(* CODESYS project MC516.project
   CompiledLibraryCompatibilityVersion: LeadSysStudio V3.5 SP15 Patch 4
   Title: MC516

Project tree, tasks and I/O mapping:
  Device : MC516, Leadshine Technology Co., Ltd., order no. 516101, version 3.5.15.40
      settings: RetainMode = 0; RetainStartAddr = 20480; RetainEndAddr = 524288; RetainSize = 524288
    application Application
      libraries: Standard, * (System)
      task EtherCAT_Master_Leadshine_A (cyclic, interval 2000 µs, priority 0) calls EtherCAT_Master_Leadshine_A.EtherCAT_Task, MAIN
      program MAIN [ST]: io, motion, save_check, save_apply, work
      DataMain/
        data type HMIData
        data type SaveData
      function block AxisFB [ST]
      Enum/
        data type State
      Object/
        data type Button
        data type Cylinder
        data type AxisEC
      function StateNext [ST]
      DataWork/
        data type SupplyData
        data type WorkData
        data type CutData
      function block CutFB [ST]
      visualisation Visualization
      function block SupplyFB [ST]
      Symbols
      global variables PersistentVars
    Resource Usage
    Device Diagnose
    Network Configuration
      LocalBus Config
    SoftMotion General Axis Pool
      JogEncoder : SMC_FreeEncoder, 3S - Smart Software Solutions GmbH, order no. 1805, version 3.5.5.0
          settings: wDriveID = 3; dwRatioTechUnitsDenom = 400; ScalingIncs = 400
    High_Speed_IO_Module : High Speed IO, Leadshine Technology Co., Ltd., version 3.5.15.40
        settings: HS_IO_Mode_0.High In IO Mode 0 = 196611; HS_IO_Mode_0.High In IO Mode 2 = 196611; Counter_Mask = 5; Ioin_Mask = 19; HS counter 1.Counter_CountMode = 1; HS counter 2.Counter_CountMode = 1; HS counter 3.Counter_SetWorkMode = 2; HS counter 3.Counter_CountMode = 1; InputFilter Para.Time_In0 = 2; InputFilter Para.Time_In1 = 2; InputFilter Para.Time_In4 = 2
        unmapped channels: Genral_IO_IN, Genral_IO_Out
    LocalBus_Master_Module : LocalBus Master, Leadshine Technology Co., Ltd., version 3.5.15.40
    EtherCAT_Master_Leadshine_A : EtherCAT Master SoftMotion, 3S - Smart Software Solutions GmbH, version 3.5.15.30
        settings: MasterCycleTime = 2000; NetworkName = 'ecat'; SelectNetworkByName = TRUE; SrcAddress1 = 10; SrcAddress2 = 889192738
      XINJE_DS5C1_CoE_Drive_Rev4_0 : XINJE-DS5C1 EtherCAT(CoE) Drive Rev4.0 v3.7.70, Xinje Electronics, Inc., order no. XINJE-DS5C1 CoE Drive Rev4.0, version Revision=16#20201207
          settings: Number of Inputs = 6; Number of Infos about Inputs = 6; StationAlias = 1; Sync.Length = 17; FMMU.Length = 17; DC sync0 cycletime = 2000; DC sync1 cycletime = 2000; Number of SDO = 4; Interpolation time period.Value = 2; RxTxPdo.NumberofEntries = 6; RxTxPdo.Index = 16#1A00; RxTxPdo.DependOnSlot = False; RxTxPdo.DependOnSlotGroup = False; RxTxPdo.OverwrittenByModule = False; Status Word.Offset = 0; Status Word.DependOnSlot = False; Status Word.DependOnSlotGroup = False; ActualPosition.Offset = 0; ActualPosition.DependOnSlot = False; ActualPosition.DependOnSlotGroup = False; Velocity actual value.Offset = 0; Velocity actual value.DependOnSlot = False; Velocity actual value.DependOnSlotGroup = False; ActualTorque.Offset = 0; ActualTorque.DependOnSlot = False; ActualTorque.DependOnSlotGroup = False; ModeOfOperationDisplay.Offset = 0; ModeOfOperationDisplay.DependOnSlot = False; ModeOfOperationDisplay.DependOnSlotGroup = False; Index = 16#5000; SubIndex = 0; Size = 32; Offset = 0; DependOnSlot = False; DependOnSlotGroup = False; Status Word.Default = ''; Status Word.Comment = ''; ActualPosition.Default = ''; ActualPosition.Comment = ''; Velocity actual value.Default = '';
            Velocity actual value.Comment = ''; ActualTorque.Default = ''; ActualTorque.Comment = ''; ModeOfOperationDisplay.Default = ''; ModeOfOperationDisplay.Comment = ''; Name = 'Encode Single Position'; DataType = 'DINT'; Default = ''; Comment = ''
          unmapped channels: Control Word, TargetPosition, TargetVelocity, TargetTorque, ModeOfOperation, Status Word, ActualPosition, Velocity actual value, ActualTorque, ModeOfOperationDisplay, Encode Single Position
        Axis : Axis, 3S - Smart Software Solutions GmbH, order no. 0, version 4.6.1.0
            settings: wDriveID = 0; dwRatioTechUnitsDenom = 16384; iRatioTechUnitsNum = -625; eRampType = 3; Number of pulses for one revolution = 131072; The displacement for one revolution of the workbench = 5000; Gear ratio molecule = 1; Gear ratio denominator = 1; ScalingIncs = 131072; InvertDirection = True; AdrOffset_8010 = 4; BitOffset_8010 = 0; BitLength_8010 = 16; Address_8010 = '%QW2'; Type_8010 = 'UINT'; AddressPointer_8010 = ADR(%QW2); AdrOffset_8020 = 8; BitOffset_8020 = 0; BitLength_8020 = 32; Address_8020 = '%QD2'; Type_8020 = 'DINT'; AddressPointer_8020 = ADR(%QD2); AdrOffset_8030 = 12; BitOffset_8030 = 0; BitLength_8030 = 32; Address_8030 = '%QD3'; Type_8030 = 'DINT'; AddressPointer_8030 = ADR(%QD3); AdrOffset_8040 = 16; BitOffset_8040 = 0; BitLength_8040 = 16; Address_8040 = '%QW8'; Type_8040 = 'INT'; AddressPointer_8040 = ADR(%QW8); AdrOffset_8050 = 18; BitOffset_8050 = 0; BitLength_8050 = 8; Address_8050 = '%QB18'; Type_8050 = 'SINT'; AddressPointer_8050 = ADR(%QB18);
              AdrOffset_8060 = 4294967295; BitOffset_8060 = 0; BitLength_8060 = 0; Address_8060 = ''; Type_8060 = ''; AddressPointer_8060 = 0; AdrOffset_8070 = 4294967295; BitOffset_8070 = 0; BitLength_8070 = 0; Address_8070 = ''; Type_8070 = ''; AddressPointer_8070 = 0; AdrOffset_8080 = 4294967295; BitOffset_8080 = 0; BitLength_8080 = 0; Address_8080 = ''; Type_8080 = ''; AddressPointer_8080 = 0; AdrOffset_8090 = 4294967295; BitOffset_8090 = 0; BitLength_8090 = 0; Address_8090 = ''; Type_8090 = ''; AddressPointer_8090 = 0; AdrOffset_8510 = 4; BitOffset_8510 = 0; BitLength_8510 = 16; Address_8510 = '%IW2'; Type_8510 = 'UINT'; AddressPointer_8510 = ADR(%IW2); AdrOffset_8520 = 8; BitOffset_8520 = 0; BitLength_8520 = 32; Address_8520 = '%ID2'; Type_8520 = 'DINT'; AddressPointer_8520 = ADR(%ID2); AdrOffset_8530 = 12; BitOffset_8530 = 0; BitLength_8530 = 32; Address_8530 = '%ID3';
              Type_8530 = 'DINT'; AddressPointer_8530 = ADR(%ID3); AdrOffset_8540 = 16; BitOffset_8540 = 0; BitLength_8540 = 16; Address_8540 = '%IW8'; Type_8540 = 'INT'; AddressPointer_8540 = ADR(%IW8); AdrOffset_8550 = 18; BitOffset_8550 = 0; BitLength_8550 = 8; Address_8550 = '%IB18'; Type_8550 = 'SINT'; AddressPointer_8550 = ADR(%IB18); AdrOffset_8560 = 4294967295; BitOffset_8560 = 0; BitLength_8560 = 0; Address_8560 = ''; Type_8560 = ''; AddressPointer_8560 = 0; AdrOffset_8570 = 4294967295; BitOffset_8570 = 0; BitLength_8570 = 0; Address_8570 = ''; Type_8570 = ''; AddressPointer_8570 = 0; AdrOffset_8580 = 4294967295; BitOffset_8580 = 0; BitLength_8580 = 0; Address_8580 = ''; Type_8580 = ''; AddressPointer_8580 = 0; AdrOffset_8590 = 4294967295; BitOffset_8590 = 0; BitLength_8590 = 0; Address_8590 = ''; Type_8590 = ''; AddressPointer_8590 = 0; AdrOffset_8600 = 4294967295; BitOffset_8600 = 0;
              BitLength_8600 = 0; Address_8600 = ''; Type_8600 = ''; AddressPointer_8600 = 0; AdrOffset_8600 = 4294967295; BitOffset_8600 = 0; BitLength_8600 = 0; Address_8610 = ''; Type_8610 = ''; AddressPointer_8610 = 0; AdrOffset_8620 = 4294967295; BitOffset_8620 = 0; BitLength_8620 = 0; Address_8620 = ''; Type_8620 = ''; AddressPointer_8620 = 0
      XINJE_DS5C1_CoE_Drive_Rev4_0_1 : XINJE-DS5C1 EtherCAT(CoE) Drive Rev4.0 v3.7.70, Xinje Electronics, Inc., order no. XINJE-DS5C1 CoE Drive Rev4.0, version Revision=16#20201207
          settings: Number of Inputs = 6; Number of Infos about Inputs = 6; StationAlias = 1; Optional = False; DeviceIdenticationADO = 0; DeviceIdenticationMode = 0; Sync.Length = 17; FMMU.Length = 17; DC sync0 cycletime = 2000; DC sync1 cycletime = 2000; Number of SDO = 4; Interpolation time period.Value = 2; RxTxPdo.NumberofEntries = 6; RxTxPdo.Index = 16#1A00; RxTxPdo.DependOnSlot = False; RxTxPdo.DependOnSlotGroup = False; RxTxPdo.OverwrittenByModule = False; Status Word.Offset = 0; Status Word.DependOnSlot = False; Status Word.DependOnSlotGroup = False; ActualPosition.Offset = 0; ActualPosition.DependOnSlot = False; ActualPosition.DependOnSlotGroup = False; Velocity actual value.Offset = 0; Velocity actual value.DependOnSlot = False; Velocity actual value.DependOnSlotGroup = False; ActualTorque.Offset = 0; ActualTorque.DependOnSlot = False; ActualTorque.DependOnSlotGroup = False; ModeOfOperationDisplay.Offset = 0; ModeOfOperationDisplay.DependOnSlot = False; ModeOfOperationDisplay.DependOnSlotGroup = False; Index = 16#5000; SubIndex = 0; Size = 32; Offset = 0; DependOnSlot = False; DependOnSlotGroup = False; Status Word.Default = ''; Status Word.Comment = '';
            ActualPosition.Default = ''; ActualPosition.Comment = ''; Velocity actual value.Default = ''; Velocity actual value.Comment = ''; ActualTorque.Default = ''; ActualTorque.Comment = ''; ModeOfOperationDisplay.Default = ''; ModeOfOperationDisplay.Comment = ''; Name = 'Encode Single Position'; DataType = 'DINT'; Default = ''; Comment = ''
          unmapped channels: Control Word, TargetPosition, TargetVelocity, TargetTorque, ModeOfOperation, Status Word, ActualPosition, Velocity actual value, ActualTorque, ModeOfOperationDisplay, Encode Single Position
        Axis_1 : Axis, 3S - Smart Software Solutions GmbH, order no. 0, version 4.6.1.0
            settings: dwRatioTechUnitsDenom = 16384; iRatioTechUnitsNum = -625; eRampType = 3; Number of pulses for one revolution = 131072; The displacement for one revolution of the workbench = 5000; Gear ratio molecule = 1; Gear ratio denominator = 1; ScalingIncs = 131072; InvertDirection = True; AdrOffset_8010 = 20; BitOffset_8010 = 0; BitLength_8010 = 16; Address_8010 = '%QW10'; Type_8010 = 'UINT'; AddressPointer_8010 = ADR(%QW10); AdrOffset_8020 = 24; BitOffset_8020 = 0; BitLength_8020 = 32; Address_8020 = '%QD6'; Type_8020 = 'DINT'; AddressPointer_8020 = ADR(%QD6); AdrOffset_8030 = 28; BitOffset_8030 = 0; BitLength_8030 = 32; Address_8030 = '%QD7'; Type_8030 = 'DINT'; AddressPointer_8030 = ADR(%QD7); AdrOffset_8040 = 32; BitOffset_8040 = 0; BitLength_8040 = 16; Address_8040 = '%QW16'; Type_8040 = 'INT'; AddressPointer_8040 = ADR(%QW16); AdrOffset_8050 = 34; BitOffset_8050 = 0; BitLength_8050 = 8; Address_8050 = '%QB34'; Type_8050 = 'SINT'; AddressPointer_8050 = ADR(%QB34); AdrOffset_8060 = 4294967295;
              BitOffset_8060 = 0; BitLength_8060 = 0; Address_8060 = ''; Type_8060 = ''; AddressPointer_8060 = 0; AdrOffset_8070 = 4294967295; BitOffset_8070 = 0; BitLength_8070 = 0; Address_8070 = ''; Type_8070 = ''; AddressPointer_8070 = 0; AdrOffset_8080 = 4294967295; BitOffset_8080 = 0; BitLength_8080 = 0; Address_8080 = ''; Type_8080 = ''; AddressPointer_8080 = 0; AdrOffset_8090 = 4294967295; BitOffset_8090 = 0; BitLength_8090 = 0; Address_8090 = ''; Type_8090 = ''; AddressPointer_8090 = 0; AdrOffset_8510 = 24; BitOffset_8510 = 0; BitLength_8510 = 16; Address_8510 = '%IW12'; Type_8510 = 'UINT'; AddressPointer_8510 = ADR(%IW12); AdrOffset_8520 = 28; BitOffset_8520 = 0; BitLength_8520 = 32; Address_8520 = '%ID7'; Type_8520 = 'DINT'; AddressPointer_8520 = ADR(%ID7); AdrOffset_8530 = 32; BitOffset_8530 = 0; BitLength_8530 = 32; Address_8530 = '%ID8'; Type_8530 = 'DINT';
              AddressPointer_8530 = ADR(%ID8); AdrOffset_8540 = 36; BitOffset_8540 = 0; BitLength_8540 = 16; Address_8540 = '%IW18'; Type_8540 = 'INT'; AddressPointer_8540 = ADR(%IW18); AdrOffset_8550 = 38; BitOffset_8550 = 0; BitLength_8550 = 8; Address_8550 = '%IB38'; Type_8550 = 'SINT'; AddressPointer_8550 = ADR(%IB38); AdrOffset_8560 = 4294967295; BitOffset_8560 = 0; BitLength_8560 = 0; Address_8560 = ''; Type_8560 = ''; AddressPointer_8560 = 0; AdrOffset_8570 = 4294967295; BitOffset_8570 = 0; BitLength_8570 = 0; Address_8570 = ''; Type_8570 = ''; AddressPointer_8570 = 0; AdrOffset_8580 = 4294967295; BitOffset_8580 = 0; BitLength_8580 = 0; Address_8580 = ''; Type_8580 = ''; AddressPointer_8580 = 0; AdrOffset_8590 = 4294967295; BitOffset_8590 = 0; BitLength_8590 = 0; Address_8590 = ''; Type_8590 = ''; AddressPointer_8590 = 0; AdrOffset_8600 = 4294967295; BitOffset_8600 = 0; BitLength_8600 = 0;
              Address_8600 = ''; Type_8600 = ''; AddressPointer_8600 = 0; AdrOffset_8600 = 4294967295; BitOffset_8600 = 0; BitLength_8600 = 0; Address_8610 = ''; Type_8610 = ''; AddressPointer_8610 = 0; AdrOffset_8620 = 4294967295; BitOffset_8620 = 0; BitLength_8620 = 0; Address_8620 = ''; Type_8620 = ''; AddressPointer_8620 = 0
      XINJE_DS5C1_CoE_Drive_Rev4_0_2 : XINJE-DS5C1 EtherCAT(CoE) Drive Rev4.0 v3.7.70, Xinje Electronics, Inc., order no. XINJE-DS5C1 CoE Drive Rev4.0, version Revision=16#20201207
          settings: Number of Inputs = 6; Number of Infos about Inputs = 6; StationAlias = 1; Optional = False; DeviceIdenticationADO = 0; DeviceIdenticationMode = 0; Sync.Length = 17; FMMU.Length = 17; DC sync0 cycletime = 2000; DC sync1 cycletime = 2000; Number of SDO = 7; Interpolation time period.Value = 2; RxTxPdo.NumberofEntries = 6; RxTxPdo.Index = 16#1A00; RxTxPdo.DependOnSlot = False; RxTxPdo.DependOnSlotGroup = False; RxTxPdo.OverwrittenByModule = False; Status Word.Offset = 0; Status Word.DependOnSlot = False; Status Word.DependOnSlotGroup = False; ActualPosition.Offset = 0; ActualPosition.DependOnSlot = False; ActualPosition.DependOnSlotGroup = False; Velocity actual value.Offset = 0; Velocity actual value.DependOnSlot = False; Velocity actual value.DependOnSlotGroup = False; ActualTorque.Offset = 0; ActualTorque.DependOnSlot = False; ActualTorque.DependOnSlotGroup = False; ModeOfOperationDisplay.Offset = 0; ModeOfOperationDisplay.DependOnSlot = False; ModeOfOperationDisplay.DependOnSlotGroup = False; Index = 16#5000; SubIndex = 0; Size = 32; Offset = 0; DependOnSlot = False; DependOnSlotGroup = False; Status Word.Default = ''; Status Word.Comment = '';
            ActualPosition.Default = ''; ActualPosition.Comment = ''; Velocity actual value.Default = ''; Velocity actual value.Comment = ''; ActualTorque.Default = ''; ActualTorque.Comment = ''; ModeOfOperationDisplay.Default = ''; ModeOfOperationDisplay.Comment = ''; Name = 'Encode Single Position'; DataType = 'DINT'; Default = ''; Comment = ''
          unmapped channels: Control Word, TargetPosition, TargetVelocity, TargetTorque, ModeOfOperation, Status Word, ActualPosition, Velocity actual value, ActualTorque, ModeOfOperationDisplay, Encode Single Position
        Axis_2 : Axis, 3S - Smart Software Solutions GmbH, order no. 0, version 4.6.1.0
            settings: wDriveID = 2; dwRatioTechUnitsDenom = 90112; iRatioTechUnitsNum = -5625; iMovementType = 0; fPositionPeriod = 360000; eRampType = 3; Number of pulses for one revolution = 131072; The displacement for one revolution of the workbench = 360000; Gear ratio molecule = 44; Gear ratio denominator = 1; ScalingIncs = 131072; ScalingMotorTurns2 = 44; InvertDirection = True; AdrOffset_8010 = 36; BitOffset_8010 = 0; BitLength_8010 = 16; Address_8010 = '%QW18'; Type_8010 = 'UINT'; AddressPointer_8010 = ADR(%QW18); AdrOffset_8020 = 40; BitOffset_8020 = 0; BitLength_8020 = 32; Address_8020 = '%QD10'; Type_8020 = 'DINT'; AddressPointer_8020 = ADR(%QD10); AdrOffset_8030 = 44; BitOffset_8030 = 0; BitLength_8030 = 32; Address_8030 = '%QD11'; Type_8030 = 'DINT'; AddressPointer_8030 = ADR(%QD11); AdrOffset_8040 = 48; BitOffset_8040 = 0; BitLength_8040 = 16; Address_8040 = '%QW24'; Type_8040 = 'INT'; AddressPointer_8040 = ADR(%QW24); AdrOffset_8050 = 50; BitOffset_8050 = 0; BitLength_8050 = 8;
              Address_8050 = '%QB50'; Type_8050 = 'SINT'; AddressPointer_8050 = ADR(%QB50); AdrOffset_8060 = 4294967295; BitOffset_8060 = 0; BitLength_8060 = 0; Address_8060 = ''; Type_8060 = ''; AddressPointer_8060 = 0; AdrOffset_8070 = 4294967295; BitOffset_8070 = 0; BitLength_8070 = 0; Address_8070 = ''; Type_8070 = ''; AddressPointer_8070 = 0; AdrOffset_8080 = 4294967295; BitOffset_8080 = 0; BitLength_8080 = 0; Address_8080 = ''; Type_8080 = ''; AddressPointer_8080 = 0; AdrOffset_8090 = 4294967295; BitOffset_8090 = 0; BitLength_8090 = 0; Address_8090 = ''; Type_8090 = ''; AddressPointer_8090 = 0; AdrOffset_8510 = 44; BitOffset_8510 = 0; BitLength_8510 = 16; Address_8510 = '%IW22'; Type_8510 = 'UINT'; AddressPointer_8510 = ADR(%IW22); AdrOffset_8520 = 48; BitOffset_8520 = 0; BitLength_8520 = 32; Address_8520 = '%ID12'; Type_8520 = 'DINT'; AddressPointer_8520 = ADR(%ID12); AdrOffset_8530 = 52;
              BitOffset_8530 = 0; BitLength_8530 = 32; Address_8530 = '%ID13'; Type_8530 = 'DINT'; AddressPointer_8530 = ADR(%ID13); AdrOffset_8540 = 56; BitOffset_8540 = 0; BitLength_8540 = 16; Address_8540 = '%IW28'; Type_8540 = 'INT'; AddressPointer_8540 = ADR(%IW28); AdrOffset_8550 = 58; BitOffset_8550 = 0; BitLength_8550 = 8; Address_8550 = '%IB58'; Type_8550 = 'SINT'; AddressPointer_8550 = ADR(%IB58); AdrOffset_8560 = 4294967295; BitOffset_8560 = 0; BitLength_8560 = 0; Address_8560 = ''; Type_8560 = ''; AddressPointer_8560 = 0; AdrOffset_8570 = 4294967295; BitOffset_8570 = 0; BitLength_8570 = 0; Address_8570 = ''; Type_8570 = ''; AddressPointer_8570 = 0; AdrOffset_8580 = 4294967295; BitOffset_8580 = 0; BitLength_8580 = 0; Address_8580 = ''; Type_8580 = ''; AddressPointer_8580 = 0; AdrOffset_8590 = 4294967295; BitOffset_8590 = 0; BitLength_8590 = 0; Address_8590 = ''; Type_8590 = '';
              AddressPointer_8590 = 0; AdrOffset_8600 = 4294967295; BitOffset_8600 = 0; BitLength_8600 = 0; Address_8600 = ''; Type_8600 = ''; AddressPointer_8600 = 0; AdrOffset_8600 = 4294967295; BitOffset_8600 = 0; BitLength_8600 = 0; Address_8610 = ''; Type_8610 = ''; AddressPointer_8610 = 0; AdrOffset_8620 = 4294967295; BitOffset_8620 = 0; BitLength_8620 = 0; Address_8620 = ''; Type_8620 = ''; AddressPointer_8620 = 0
  text list GlobalTextList
*)

// Device/Application/DataMain/HMIData
{ attribute 'pack_mode' := ''}
TYPE HMIData :
STRUCT
	//
	save_data: SaveData;
	save: BOOL;
	save_need_check: BOOL;
	save_need: BOOL;
	//
	plc_ready: BOOL;
	hmi_ready: BOOL;
	run: BOOL;
	stop: BOOL;
	home: BOOL;
	overload_fixed: BOOL;
	foil_stuck_fix: BOOL;
	//
	supply_test: BOOL;
	supply_arm_clamp_holder: BOOL;
	supply_arm_clamp: BOOL;
	supply_spindle_clamp: BOOL;
	supply_spindle_extract: BOOL;
	supply_feeder_small: BOOL;
	supply_feeder_linear: BOOL;
	supply_feeder_big: BOOL;
	supply_feeder_test: BOOL;
	cut_spindle_run: BOOL;
	hydraulic_run: BOOL;
	jog_micro_per_rev: UINT;
	//
	view_input_run: BOOL;
	view_input_stop: BOOL;
	view_input_air: BOOL;
	view_input_hydraulic: BOOL;
	view_input_arm_clamp_holder_p: BOOL;
	view_input_feeder_small: BOOL;
	view_input_feeder_big: BOOL;
	view_input_jog_counter_a: BOOL;
	view_input_jog_counter_b: BOOL;
	view_input_jog_index_a: BOOL;
	view_input_jog_index_b: BOOL;
	view_input_spindle_encoder: BOOL;
	view_input_jog_index: UINT;
	view_input_jog_micro: DINT;
	//
	view_output_arm_clamp_holder: BOOL;
	view_output_arm_clamp: BOOL;
	view_output_spindle: BOOL;
	view_output_spindle_clamp_n: BOOL;
	view_output_spindle_clamp_p: BOOL;
	view_output_spindle_extract: BOOL;
	view_output_hydraulic: BOOL;
	view_output_alarm: BOOL;
	view_output_feeder_small: BOOL;
	view_output_feeder_linear: BOOL;
	view_output_feeder_big: BOOL;
	//
	view_can_run: BOOL;
	view_can_stop: BOOL;
	view_can_home: BOOL;
	view_run_auto: BOOL;
	view_manual_active: BOOL;
	//
	view_axiss_position_micron: ARRAY[0..2] OF UDINT;
	view_axiss_torque_mNm: ARRAY[0..2] OF UDINT;
	view_cut_spindle_run_ing: BOOL;
	view_cut_spindle_rpm: UDINT;
	//
	view_supply_test: ARRAY[0..4] OF BOOL;
	//
	view_overload: BOOL;
	view_supply_foil_short: BOOL;
	view_supply_foil_stuck: BOOL;
	view_cycle_count: UDINT;
	view_cycle_time_msec: UDINT;
	//
	view_state_work: INT;
	view_state_supply: INT;
	view_state_cut: INT;
	view_state_cut_spindle: INT;
END_STRUCT
END_TYPE

// Device/Application/DataMain/SaveData
{ attribute 'pack_mode' := ''}
TYPE SaveData :
STRUCT
	set_done: BOOL;
	//
	supply_begin_micro_deg: UDINT;
	supply_mid_micro_deg: UDINT;
	supply_end_micro_deg: UDINT;
	supply_micro_deg_per_sec: UDINT;
	//
	supply_arm_clamp_holder_n_delay_msec: UINT;
	supply_arm_clamp_holder_p_delay_msec: UINT;
	supply_arm_clamp_n_delay_msec: UINT;
	supply_arm_clamp_p_delay_msec: UINT;
	supply_spindle_clamp_n_delay_msec: UINT;
	supply_spindle_clamp_p_delay_msec: UINT;
	supply_spindle_extract_n_delay_msec: UINT;
	supply_spindle_extract_p_delay_msec: UINT;
	//
	cut_begin_micron: ARRAY[0..1] OF UDINT;
	cut_rapid_micron: ARRAY[0..1] OF UDINT;
	cut_end_micron: ARRAY[0..1] OF UDINT;
	cut_offset_micron: ARRAY[0..1] OF DINT;
	cut_lag_micron: UDINT;
	cut_rapid_micron_per_rev: UDINT;
	cut_micron_per_rev: UDINT;
	cut_dwell_msec: UINT;
	cut_retract_micron: UDINT; // vị trí lùi về
	cut_retract_micron_per_sec: UDINT; // tốc độ lùi sau khi cắt
	cut_spindle_encoder_resolution: UINT;
	//
	home_encoder_value_recorded: BOOL;
	home_encoder_value: ARRAY[0..2] OF DINT;
END_STRUCT
END_TYPE

// Device/Application/Enum/State
{attribute 'qualified_only'}
{attribute 'strict'}
TYPE State :
(
	NONE := 0,
	RST := 1,
	RST_DONE := 50,
	HOME := 51,
	HOME_FORWARD := 71,
	HOME_DONE := 90,
	HOME_OFFSET := 91,
	HOME_OFFSET_DONE := 99,
	READY := 100,
	RUN := 101,
	RUN_ING := 200
);
END_TYPE

// Device/Application/Object/Button
{ attribute 'pack_mode' := ''}
TYPE Button :
STRUCT
	on: BOOL;
	rise: R_TRIG;
	rise_physical: R_TRIG;
	fall: F_TRIG;
	fall_physical: F_TRIG;
	timer: TON;
END_STRUCT
END_TYPE

// Device/Application/Object/Cylinder
{ attribute 'pack_mode' := ''}
TYPE Cylinder :
STRUCT
	on: BOOL;
	n_timer: TON;
	p_timer: TON;
END_STRUCT
END_TYPE

// Device/Application/Object/AxisEC
{ attribute 'pack_mode' := ''}
TYPE AxisEC :
STRUCT
	///////
	//REF//
	///////
	ref: POINTER TO SM3_Drive_ETC_DS402_CyclicSync.AXIS_REF_ETC_DS402_CS;
	read: POINTER TO SMC3_ETC_ReadParameter_CoE;
	write: POINTER TO SMC3_ETC_WriteParameter_CoE;
	read_status: POINTER TO MC_ReadStatus;
	set_mode: POINTER TO SMC_SetControllerMode;
	power: POINTER TO MC_Power;
	reset: POINTER TO MC_Reset;
	stop: POINTER TO MC_Stop;
	inch: POINTER TO SMC_Inch;
	fsv: POINTER TO SMC_FollowSetValues;
	sp: POINTER TO MC_SetPosition;
	mabs: POINTER TO MC_MoveAbsolute;
	////////
	//DATA//
	////////
	encoder_resolution: DINT;
	torque_rated_Nm: LREAL;
	encoder_single_position: DINT;
	///////////
	//PROCESS//
	///////////
	state: INT;
	torque_Nm: LREAL;
	torque_Nm_abs: LREAL;
	overload: BOOL;
	overload_check: BOOL;
	overload_timer: TON;
	//home
	home_done: BOOL; // = TRUE khi về gốc thành công, chỉ về gốc khi bật máy
	home_torque_Nm: LREAL;
	home_hit_timer: TON;
	home_offset_absolute_μ: LREAL; // vị trí từ điểm va chạm đến gốc tuyệt đối, xem hàm save_apply()
	home_back_μ_per_sec: LREAL; // tốc độ lùi về lấy gốc
	home_forward_μ_per_sec: LREAL; // tốc độ tiến sau khi lấy gốc xong
	home_offset_μ: LREAL; // giá trị này để thực hiện lệnh state = State.HOME_OFFSET ở trong AxisLinearFB
	home_encoder_value_recorded: BOOL;
	home_encoder_value: POINTER TO DINT; // pointer tới giá trị ở save data
	home_encoder_delta: DINT;
	home_delta_μ: LREAL;
	//
	ramp_time_sec: LREAL;
	jerk_factor: LREAL;
	//
	jog_delta: LREAL;
	jog_velocity: LREAL;
	jog_acceleration: LREAL;
	max_μ: LREAL; // giới hạn vị trí tối đa có thể di chuyển từ gốc tuyệt đối
	max_μ_per_sec: LREAL; // giới hạn tốc độ tối đa
	//run
	target_position_μ: LREAL; // sử dụng cho state = State.RUN ở trong AxisLinearFB
	target_velocity_μ_per_sec: LREAL; // sử dụng cho state = State.RUN ở trong AxisLinearFB
END_STRUCT
END_TYPE

// Device/Application/DataWork/SupplyData
{ attribute 'pack_mode' := ''}
TYPE SupplyData :
STRUCT
	state: INT;
	axis: AxisEC;
	axis_fb: AxisFB;
	state_ready: BOOL;
	//
	input_air: BOOL;
	input_hydraulic: BOOL;
	input_arm_clamp_holder_p: BOOL;
	input_feeder_small: BOOL;
	input_feeder_big: BOOL;
	hydraulic: BOOL;
	feeder_small: BOOL;
	feeder_small_on_timer: TON;
	feeder_small_off_timer: TON;
	feeder_linear: BOOL;
	feeder_big: BOOL;
	feeder_test: BOOL;
	arm_clamp_holder: Cylinder;
	arm_clamp_holder_p_rise: R_TRIG;
	arm_clamp: Cylinder;
	spindle_clamp: Cylinder;
	spindle_clamp_release: BOOL;
	spindle_extract: Cylinder;
	//
	begin_μdeg: LREAL;
	mid_μdeg: LREAL;
	end_μdeg: LREAL;
	μdeg_per_sec: LREAL;
	foil_short: BOOL;
	foil_short_rise: R_TRIG;
	foil_stuck: BOOL;
	foil_stuck_timer: TON;
	foil_stuck_fix_rise: R_TRIG;
	foil_stuck_fix_timer: TON;
END_STRUCT
END_TYPE

// Device/Application/DataWork/WorkData
{ attribute 'pack_mode' := ''}
TYPE WorkData :
STRUCT
	state: INT;
	//
	input_run: Button;
	input_stop: Button;
	input_home: Button;
	input_jog_index: UINT;
	//
	can_run: BOOL;
	can_stop: BOOL;
	can_home: BOOL;
	jog_i: POINTER TO AxisEC;
	jog_encoder_counter: LS_Counter;
	jog_encoder_counter_set: LS_PresetValue;
	jog_encoder: POINTER TO SM3_Basic.FREE_ENCODER_REF;
	jog_encoder_last: LREAL;
	run_auto: Button;
	overload: BOOL;
	overload_rise: R_TRIG;
	overload_fixed_rise: R_TRIG;
	alarm: BOOL;
	//
	cut_spindle_run_rise: R_TRIG;
	cut_spindle_run_timer: TON;
	supply_hydraulic_rise: R_TRIG;
	supply_hydraulic_timer: TON;
	supply_test_timer: TON;
	//
	manual_active: BOOL;
	final_cycle_flag: BOOL;
	final_cycle: BOOL;
	cycle_start_msec: ULINT;
	cycle_time_msec: UDINT;
END_STRUCT
END_TYPE

// Device/Application/DataWork/CutData
{ attribute 'pack_mode' := ''}
TYPE CutData :
STRUCT
	state: INT;
	axiss: ARRAY[0..1] OF AxisEC;
	axiss_fb: ARRAY[0..1] OF AxisFB;
	//
	state_spindle: INT;
	spindle: BOOL;
	spindle_encoder_counter_last: DINT;
	spindle_encoder_counter: LS_Counter;
	spindle_encoder_resolution: UDINT;
	spindle_encoder_time_msec_last: ULINT;
	spindle_rps_last: LREAL;
	spindle_rps: LREAL;
	spindle_rps_stable_cycle: INT;
	time_msec: ULINT;
	time_delta_sec: LREAL;
	//
	begin_μm: ARRAY[0..1] OF LREAL;
	rapid_μm: ARRAY[0..1] OF LREAL;
	end_μm: ARRAY[0..1] OF LREAL;
	lag_μm: LREAL;
	rapid_μm_per_rev: LREAL;
	μm_per_rev: LREAL;
	dwell_timer: TON;
	retract_μm: LREAL;
	retract_μm_per_sec: LREAL;
END_STRUCT
END_TYPE

// Device/Application/PersistentVars
{attribute 'qualified_only'}
VAR_GLOBAL PERSISTENT RETAIN
END_VAR
VAR_GLOBAL PERSISTENT
	MAIN.save_data: SaveData;
END_VAR

// Device/Application/MAIN
PROGRAM MAIN
VAR
	time_msec_last: ULINT;
	time_msec : ULINT;
	time_delta_sec: LREAL;
	//
	axiss: ARRAY [0..2] OF POINTER TO SM3_Drive_ETC_DS402_CyclicSync.AXIS_REF_ETC_DS402_CS;
	// dùng pointer để dễ dàng thao tác với nhiều trục hơn, xem hàm motion()
	axiss_read: ARRAY[0..2] OF SMC3_ETC_ReadParameter_CoE;
	axiss_write: ARRAY[0..2] OF SMC3_ETC_WriteParameter_CoE;
	axiss_read_status: ARRAY[0..2] OF MC_ReadStatus;
	axiss_set_mode: ARRAY[0..2] OF SMC_SetControllerMode;
	axiss_power: ARRAY[0..2] OF MC_Power; // bật tắt động cơ
	axiss_reset: ARRAY[0..2] OF MC_Reset; // reset lỗi
	axiss_stop: ARRAY[0..2] OF MC_Stop; // dừng
	axiss_inch: ARRAY[0..2] OF SMC_Inch;
	axiss_fsv: ARRAY[0..2] OF SMC_FollowSetValues;
	axiss_sp: ARRAY[0..2] OF MC_SetPosition;
	axiss_mabs: ARRAY[0..2] OF MC_MoveAbsolute;
	axiss_encoder_resolution: ARRAY[0..2] OF DINT;
	axiss_rated_torque_Nm: ARRAY[0..2] OF LREAL;
	axiss_ready: BOOL;
	//
	state_main: INT;
	main_save: Button;
	supply_data: SupplyData;
	supply_fb: SupplyFB;
	cut_data: CutData;
	cut_fb: CutFB;
	work_data: WorkData;
	hmi_data: HMIData;
	//
	i: UINT;
	j: UINT;
	k: UINT;
	axis_ec_i: POINTER TO AxisEC;
	axis_fb_i: POINTER TO AxisFB;
	//
	udint_min: UDINT;
	udint_max: UDINT;
	//
	test: BOOL;
END_VAR

VAR CONSTANT
	c_axis_count: UINT := 3;
	c_axis_i_max: UINT := c_axis_count - 1;
	c_supply_μdeg_max: UDINT := 108_000;
	c_supply_μdeg_per_sec_max: LREAL := (3000 / (60 * 42)) * 360_000; // 3000 rpm, 5_000 μdeg 1 vòng
	c_cut_stroke_μm: UDINT := 56_000;
	c_cut_μm_per_sec_max: LREAL := (3000 / 60) * 5_000; // 3000 rpm, 5_000 μm 1 vòng
END_VAR

VAR RETAIN
	cycle_count: UDINT;
	cycle_count_reset_time_msec: ULINT;
END_VAR

VAR PERSISTENT
	save_data: SaveData;
END_VAR

MC_SysLib.SysTimeRtc.SysTimeRtcHighResGet(pTimestamp:= time_msec);
time_delta_sec := ULINT_TO_LREAL(time_msec - time_msec_last) * 1E-3;
time_msec_last := time_msec;
IF state_main > 10 THEN
	motion();
	// chạy hàm motion(), vì state 11 trở đi có đoạn đọc dữ liệu của Servo
	// mà hàm motion() này lại bao gồm tất cả các lệnh của Servo
	// có thể thay đổi logic đoạn này nhưng không cần thiết lắm
END_IF
CASE state_main OF
	State.NONE: // khi khởi động thì state_main = 0 tức là = State.NONE
		test := FALSE;
		axiss[0] := ADR(Axis); // k = ADR(x) viết tắt cho "address of x" là hàm để lấy giá trị con trỏ (pointer) về biến x
		axiss[1] := ADR(Axis_1); // ví dụ muốn thay đổi giá trị của x ta sẽ viết k^ = 12345
		axiss[2] := ADR(Axis_2);
		work_data.jog_encoder := ADR(JogEncoder);
		StateNext(state_main); // chuyển tới trạng thái tiếp theo
	1:
		FOR i := 0 TO c_axis_i_max BY 1 DO // hàm FOR, FOR i = 0 TO 3 BY 1 DO sẽ chạy 4 lần i = [0, 1, 2, 3]
			CASE i OF // hàm CASE, lựa chọn theo giá trị i
				0:
					axis_ec_i := ADR(cut_data.axiss[0]);
					axis_fb_i := ADR(cut_data.axiss_fb[0]);
				1:
					axis_ec_i := ADR(cut_data.axiss[1]);
					axis_fb_i := ADR(cut_data.axiss_fb[1]);
				2:
					axis_ec_i := ADR(supply_data.axis);
					axis_fb_i := ADR(supply_data.axis_fb);
			END_CASE
			axis_ec_i^.ref := axiss[i];
			axis_ec_i^.read := ADR(axiss_read[i]);
			axis_ec_i^.write := ADR(axiss_write[i]);
			axis_ec_i^.read_status := ADR(axiss_read_status[i]);
			axis_ec_i^.set_mode := ADR(axiss_set_mode[i]);
			axis_ec_i^.power := ADR(axiss_power[i]);
			axis_ec_i^.reset := ADR(axiss_reset[i]);
			axis_ec_i^.stop := ADR(axiss_stop[i]);
			axis_ec_i^.inch := ADR(axiss_inch[i]);
			axis_ec_i^.fsv := ADR(axiss_fsv[i]);
			axis_ec_i^.sp := ADR(axiss_sp[i]);
			axis_ec_i^.mabs := ADR(axiss_mabs[i]);
			axis_fb_i^.data := axis_ec_i;
		END_FOR
		StateNext(state_main);
	2:
		axiss_ready := TRUE; // biến tạm thời để kiểm tra tất cả các servo đã hoàn thành lệnh hay chưa
		FOR i := 0 TO c_axis_i_max BY 1 DO
			IF axiss[i]^.wCommunicationState <> 100 THEN
				// nếu trạng thái wCommunicationState của servo bất kỳ không = 100 thì
				// chứng tỏ chưa hoàn thành kết nối tất cả các servo, nên ta cho giá trị axiss_ready := FALSE
				axiss_ready := FALSE;
			END_IF
		END_FOR
		IF axiss_ready THEN // hoàn thành kết nối tất cả servo, ta đên bước tiếp theo
			state_main := 11;
		END_IF
	11:
		FOR i := 0 TO c_axis_i_max BY 1 DO
			// bật động cơ, phải đặt ba biến của hàm MC_Power này = TRUE
			axiss_power[i].Enable := TRUE;
			axiss_power[i].bDriveStart := TRUE;
			axiss_power[i].bRegulatorOn := TRUE;
		END_FOR
		StateNext(state_main);
	12:
		axiss_ready := TRUE;
		FOR i := 0 TO c_axis_i_max BY 1 DO
			IF NOT axiss_power[i].Status THEN // axiss_power[i].Status = TRUE tức là đã bật Servo thành công
				axiss_ready := FALSE;
			END_IF
		END_FOR
		IF axiss_ready THEN
			StateNext(state_main);
		END_IF
	13: // đọc dữ liệu từ servo
		FOR i := 0 TO c_axis_i_max BY 1 DO
			axiss_read[i].uiIndex := 16#608F; // mở ETHERCAT/XINJE_DS5C1.../ xem trong mục "CoE Online"
			axiss_read[i].usiSubIndex := 1; //
			axiss_read[i].xExecute := TRUE;
		END_FOR
		StateNext(state_main);
	14:
		axiss_ready := TRUE;
		FOR i := 0 TO c_axis_i_max BY 1 DO
			IF NOT axiss_read[i].xDone THEN
				axiss_ready := FALSE;
			END_IF
		END_FOR
		IF axiss_ready THEN
			FOR i := 0 TO c_axis_i_max BY 1 DO
				axiss_read[i].xExecute := FALSE;
				// Sau thực hiện hàm thành công phải đặt Execute = FALSE để cho lần đọc tiếp theo
				// vì đa số hàm chỉ chạy khi Execute chuyển từ FALSE sang TRUE (Rising edge)
				// xem Defination của hàm đê biết thêm chi tiết
				axiss_encoder_resolution[i] := DWORD_TO_DINT(axiss_read[i].dwValue);
			END_FOR
			StateNext(state_main);
		END_IF
	15:
		FOR i := 0 TO c_axis_i_max BY 1 DO
			axiss_read[i].uiIndex := 16#6076;
			axiss_read[i].usiSubIndex := 0;
			axiss_read[i].xExecute := TRUE;
		END_FOR
		StateNext(state_main);
	16:
		axiss_ready := TRUE;
		FOR i := 0 TO c_axis_i_max BY 1 DO
			IF NOT axiss_read[i].xDone THEN
				axiss_ready := FALSE;
			END_IF
		END_FOR
		IF axiss_ready THEN
			FOR i := 0 TO c_axis_i_max BY 1 DO
				axiss_read[i].xExecute := FALSE;
				axiss_rated_torque_Nm[i] := DWORD_TO_LREAL(axiss_read[i].dwValue) * 1E-3;
			END_FOR
			StateNext(state_main);
		END_IF
	17:
		cut_data.axiss[0].encoder_resolution := axiss_encoder_resolution[0];
		cut_data.axiss[0].torque_rated_Nm := axiss_rated_torque_Nm[0];
		cut_data.axiss[1].encoder_resolution := axiss_encoder_resolution[1];
		cut_data.axiss[1].torque_rated_Nm := axiss_rated_torque_Nm[1];
		supply_data.axis.encoder_resolution := axiss_encoder_resolution[2];
		supply_data.axis.torque_rated_Nm := axiss_rated_torque_Nm[2];
		IF NOT save_data.set_done THEN
			save_data.set_done := TRUE;
			// biến "set_done" này nằm trong cấu trúc "save_data" nhằm mục đích
			// gán giá trị đầu cho biến lưu, đảm bảo đoạn gán dữ liệu này chỉ chạy 1 lần khi
			// PLC chạy lần dầu sau khi nạp lại chương trình.
			save_data.supply_begin_micro_deg := 10_780;
			save_data.supply_mid_micro_deg := 90_000;
			save_data.supply_end_micro_deg := 101_580;
			save_data.supply_micro_deg_per_sec := 180_000;
			//
			save_data.supply_arm_clamp_holder_n_delay_msec := 0_201;
			save_data.supply_arm_clamp_holder_p_delay_msec := 0_202;
			save_data.supply_arm_clamp_n_delay_msec := 0_203;
			save_data.supply_arm_clamp_p_delay_msec := 0_204;
			save_data.supply_spindle_clamp_n_delay_msec := 0_505;
			save_data.supply_spindle_clamp_p_delay_msec := 0_206;
			save_data.supply_spindle_extract_n_delay_msec := 0_207;
			save_data.supply_spindle_extract_p_delay_msec := 0_208;
			//
			save_data.cut_begin_micron[0] := 46_000;
			save_data.cut_begin_micron[1] := 46_000;
			save_data.cut_rapid_micron[0] := 51_000;
			save_data.cut_rapid_micron[1] := 51_000;
			save_data.cut_end_micron[0] := 53_500;
			save_data.cut_end_micron[1] := 53_500;
			save_data.cut_offset_micron[0] := -9_000;
			save_data.cut_offset_micron[1] := -9_000;
			//
			save_data.cut_lag_micron := 0_500;
			save_data.cut_rapid_micron_per_rev := 0_300; // => 0.4 * 50 = 20_000 μm/s
			save_data.cut_micron_per_rev := 0_025; // spindle 3000 rpm = 50 rps => cut_micron_per_sec = 0_2 * 50 = 10_000 μm/s
			save_data.cut_dwell_msec := 0_020;
			save_data.cut_retract_micron := 30_000;
			save_data.cut_retract_micron_per_sec := 150_000;
			save_data.cut_spindle_encoder_resolution := 1;
			//
			save_data.home_encoder_value_recorded := FALSE;
			save_data.home_encoder_value[0] := 0;
			save_data.home_encoder_value[1] := 0;
			save_data.home_encoder_value[2] := 0;
		END_IF
		StateNext(state_main);
	18:
		save_apply();
		StateNext(state_main);
	19:
		hmi_data.plc_ready := TRUE; // sau khi đã khởi động Servo bla bla thì ta PLC ready
		work_data.state := State.RST; // reset work
		state_main := State.RUN_ING; // bước vào giai đoạn chạy
		supply_fb.data := ADR(supply_data);
		cut_fb.data := ADR(cut_data);
	State.RUN_ING:
		io(); // kiểm tra io (gồm PLC io và HMI)
		supply_fb(data:= ); // hàm điều khiển cơ cấu cấp phôi (gồm servo và các xylanh khí nén)
		cut_fb(data:= ); // hàm điều khiển trục cắt
		work(); // hàm phối hợp giữa cấp phôi và cắt
END_CASE

ACTION io:
////////////
//HMI DOWN//
///////////
IF hmi_data.hmi_ready THEN
	////////
	//WORK//
	////////
	work_data.input_run.rise(CLK:= hmi_data.run, Q=> );
	work_data.input_stop.rise(CLK:= hmi_data.stop, Q=> );
	work_data.input_home.rise(CLK:= hmi_data.home, Q=> );
	work_data.overload_fixed_rise(CLK:= hmi_data.overload_fixed, Q=> );
	work_data.supply_hydraulic_rise(CLK:= hmi_data.hydraulic_run, Q=> );
	work_data.supply_hydraulic_timer(IN:= hmi_data.hydraulic_run, PT:= , Q=> , ET=> );
	work_data.supply_test_timer(IN:= hmi_data.supply_test, PT:= , Q=> , ET=> );
	work_data.cut_spindle_run_rise(CLK:= hmi_data.cut_spindle_run, Q=> );
	work_data.cut_spindle_run_timer(IN:= hmi_data.cut_spindle_run, PT:= , Q=> , ET=> );
	supply_data.foil_stuck_fix_rise(CLK:= hmi_data.foil_stuck_fix, Q=> );
	supply_data.foil_stuck_fix_timer(IN:= hmi_data.foil_stuck_fix, PT:= , Q=> , ET=> );
	////////
	//SAVE//
	////////
	IF hmi_data.save_need_check THEN
		save_check();
		hmi_data.save_need_check := FALSE;
	END_IF
	main_save.rise(CLK:= hmi_data.save, Q=> ); // Trên HMI sẽ xuất hiện nút save khi biến hmi_data.save_need = true.
	IF main_save.rise.Q THEN
		save_data := hmi_data.save_data;
		save_apply();
		hmi_data.save_need := FALSE;
		hmi_data.save := FALSE;
	END_IF
END_IF
/////////
//INPUT//
/////////
cut_data.axiss[0].encoder_single_position := DWORD_TO_DINT(%ID5);
cut_data.axiss[1].encoder_single_position := DWORD_TO_DINT(%ID10);
supply_data.axis.encoder_single_position := DWORD_TO_DINT(%ID15);
cut_data.time_msec := time_msec;
//
//jog encoder A phase %IX0.0
//jog encoder B phase %IX0.1
work_data.jog_encoder_counter(xEnable:= work_data.state = State.READY, eChannel:= COUNTER0, xValid=> , xError=> , eErrorID=> , diValue=> work_data.jog_encoder^.diEncoderPosition);
work_data.jog_encoder_counter_set(xExecute:= , eChannel:= COUNTER0, eTriggerEdge:= , diPresetValue:= , xDone=> , xBusy=> , xError=> , eErrorID=> );
work_data.input_run.rise_physical.CLK := %IX0.2;
work_data.input_stop.fall_physical.CLK := %IX0.3;
//spindle encoder %IX0.4
cut_data.spindle_encoder_counter(xEnable:= TRUE, eChannel:= COUNTER2, xValid=> , xError=> , eErrorID=> , diValue=> );
supply_data.input_feeder_small := %IX0.5;
supply_data.input_feeder_big := %IX0.6;
//empty %IX0.7
work_data.input_jog_index := (BOOL_TO_UINT(%IX1.0) +
										BOOL_TO_UINT(%IX1.1) * 2);
//empty %IX1.2 -> control panel
//empty %IX1.3 -> control panel
IF NOT test THEN
	supply_data.input_air := %IX1.4;
	supply_data.input_hydraulic := %IX1.5;
END_IF
supply_data.input_arm_clamp_holder_p := %IX1.6;
//empty %IX1.7
//
work_data.can_run := work_data.input_stop.fall_physical.CLK AND supply_data.input_air AND supply_data.input_hydraulic AND work_data.state = State.READY;
work_data.can_stop := work_data.state >= State.NONE;
work_data.can_home := work_data.state = State.RST_DONE OR work_data.state = State.READY;
IF cut_data.axiss[0].overload OR cut_data.axiss[1].overload OR supply_data.axis.overload THEN
	work_data.overload := TRUE;
END_IF
IF work_data.overload_fixed_rise.Q THEN
	cut_data.axiss[0].overload := FALSE;
	cut_data.axiss[1].overload := FALSE;
	supply_data.axis.overload := FALSE;
	cut_data.axiss[0].overload_timer.IN := FALSE;
	cut_data.axiss[1].overload_timer.IN := FALSE;
	supply_data.axis.overload_timer.IN := FALSE;
	work_data.overload := FALSE;
END_IF
//
work_data.input_run.rise_physical(CLK:= , Q=> );
work_data.input_stop.fall_physical(CLK:= , Q=> );
work_data.input_run.timer(IN:= work_data.input_run.rise.CLK OR work_data.input_run.rise_physical.CLK, PT:= , Q=> , ET=> );
work_data.run_auto.timer(IN:= work_data.input_run.rise.CLK OR work_data.input_run.rise_physical.CLK, PT:= , Q=> , ET=> );
IF work_data.input_home.rise.Q AND work_data.can_home THEN
	cut_data.axiss[0].home_done := FALSE;
	cut_data.axiss[1].home_done := FALSE;
	supply_data.axis.home_done := FALSE;
	work_data.state := State.HOME;
END_IF
IF work_data.input_stop.fall_physical.CLK AND NOT work_data.overload THEN
	IF work_data.run_auto.timer.Q THEN
		work_data.run_auto.on := TRUE;
	END_IF
	CASE work_data.state OF
		State.RST_DONE:
			IF work_data.input_run.rise.Q OR work_data.input_run.rise_physical.Q THEN
				work_data.state := State.HOME;
			END_IF
		State.READY:
			IF work_data.can_run AND supply_data.state_ready AND cut_data.state = State.READY THEN
				IF (work_data.input_run.timer.Q OR work_data.run_auto.on OR work_data.final_cycle_flag) AND cut_data.state_spindle = State.RUN_ING THEN
					IF work_data.final_cycle_flag THEN
						work_data.final_cycle_flag := FALSE;
						work_data.final_cycle := TRUE;
					END_IF
					work_data.state := State.RUN;
				END_IF
			END_IF
		ELSE
			IF work_data.run_auto.on AND (work_data.input_run.rise.Q OR work_data.input_run.rise_physical.Q) THEN
				work_data.run_auto.on := FALSE;
				work_data.final_cycle_flag := TRUE;
			END_IF
	END_CASE
END_IF
work_data.overload_rise(CLK:= work_data.overload, Q=> );
IF (work_data.input_stop.rise.Q OR work_data.input_stop.fall_physical.Q OR work_data.overload_rise.Q) AND work_data.can_stop THEN
	hmi_data.jog_micro_per_rev := 0;
	work_data.run_auto.on := FALSE;
	work_data.state := State.RST;
END_IF
IF supply_data.input_air AND supply_data.input_hydraulic AND work_data.supply_test_timer.Q THEN
	CASE supply_data.state OF
		State.READY:
			supply_data.state := State.RUN;
		110:
			supply_data.state := 111;
		120:
			supply_data.state := 121;
		130:
			supply_data.state := 131;
		140:
			supply_data.state := State.RUN;
	END_CASE
END_IF
IF supply_data.foil_stuck THEN
	IF (supply_data.state = 110 OR supply_data.state = 140) AND supply_data.foil_stuck_fix_rise.Q THEN
		supply_data.state := State.RUN; // run extract foil
	END_IF
	IF supply_data.state = 110 AND supply_data.foil_stuck_fix_timer.Q THEN
		supply_data.state := 111;
	END_IF
END_IF
IF work_data.manual_active THEN
	IF cut_data.state_spindle = State.READY AND work_data.cut_spindle_run_timer.Q THEN
		cut_data.state_spindle := State.RUN;
	END_IF
	IF cut_data.state_spindle >= State.RUN AND work_data.cut_spindle_run_rise.Q THEN
		cut_data.state_spindle := State.RST;
	END_IF
	IF NOT supply_data.hydraulic THEN
		IF work_data.supply_hydraulic_timer.Q THEN
			supply_data.hydraulic := TRUE;
		END_IF
	ELSE
		IF work_data.supply_hydraulic_rise.Q THEN
			supply_data.hydraulic := FALSE;
		END_IF
	END_IF
	IF work_data.input_run.rise.Q OR work_data.input_run.rise_physical.Q THEN
		IF supply_data.state = 110 OR supply_data.state = 120 OR supply_data.state = 130 THEN
			supply_data.state := 141;
		END_IF
		IF supply_data.state = 140 THEN
			supply_data.state := State.READY;
		END_IF
	END_IF
	IF supply_data.state = State.READY THEN
		supply_data.arm_clamp_holder.on := hmi_data.supply_arm_clamp_holder;
		supply_data.arm_clamp.on := hmi_data.supply_arm_clamp;
		supply_data.spindle_clamp.on := hmi_data.supply_spindle_clamp;
		supply_data.spindle_extract.on := hmi_data.supply_spindle_extract;
	ELSE
		hmi_data.supply_arm_clamp_holder := supply_data.arm_clamp_holder.on;
		hmi_data.supply_arm_clamp := supply_data.arm_clamp.on;
		hmi_data.supply_spindle_clamp := supply_data.spindle_clamp.on;
		hmi_data.supply_spindle_extract := supply_data.spindle_extract.on;
	END_IF
	IF supply_data.feeder_test THEN
		supply_data.feeder_small := hmi_data.supply_feeder_small;
		supply_data.feeder_linear := hmi_data.supply_feeder_linear;
		supply_data.feeder_big := hmi_data.supply_feeder_big;
	ELSE
		hmi_data.supply_feeder_small := supply_data.feeder_small;
		hmi_data.supply_feeder_linear := supply_data.feeder_linear;
		hmi_data.supply_feeder_big := supply_data.feeder_big;
	END_IF
	supply_data.feeder_test := hmi_data.supply_feeder_test;
ELSE
	hmi_data.supply_arm_clamp_holder := supply_data.arm_clamp_holder.on;
	hmi_data.supply_arm_clamp := supply_data.arm_clamp.on;
	hmi_data.supply_spindle_clamp := supply_data.spindle_clamp.on;
	hmi_data.supply_spindle_extract := supply_data.spindle_extract.on;
	hmi_data.supply_feeder_small := supply_data.feeder_small;
	hmi_data.supply_feeder_linear := supply_data.feeder_linear;
	hmi_data.supply_feeder_big := supply_data.feeder_big;
	hmi_data.supply_feeder_test := supply_data.feeder_test;
END_IF
//
supply_data.arm_clamp_holder.n_timer(IN:= NOT supply_data.arm_clamp_holder.on, PT:= , Q=> , ET=> );
supply_data.arm_clamp_holder.p_timer(IN:= supply_data.arm_clamp_holder.on, PT:= , Q=> , ET=> );
supply_data.arm_clamp.n_timer(IN:= NOT supply_data.arm_clamp.on, PT:= , Q=> , ET=> );
supply_data.arm_clamp.p_timer(IN:= supply_data.arm_clamp.on, PT:= , Q=> , ET=> );
supply_data.spindle_clamp.n_timer(IN:= NOT supply_data.spindle_clamp.on, PT:= , Q=> , ET=> );
supply_data.spindle_clamp.p_timer(IN:= supply_data.spindle_clamp.on, PT:= , Q=> , ET=> );
supply_data.spindle_extract.n_timer(IN:= NOT supply_data.spindle_extract.on, PT:= , Q=> , ET=> );
supply_data.spindle_extract.p_timer(IN:= supply_data.spindle_extract.on, PT:= , Q=> , ET=> );
//////////
//OUTPUT//
//////////
supply_data.spindle_clamp_release := (NOT supply_data.spindle_clamp.on AND NOT supply_data.spindle_clamp.n_timer.Q);
work_data.alarm := work_data.overload OR supply_data.foil_short;
%QX0.0 := supply_data.spindle_clamp.on; // relay 1
%QX0.1 := supply_data.spindle_clamp_release; // relay 2
%QX0.2 := supply_data.hydraulic; // relay 3
%QX0.3 := supply_data.arm_clamp_holder.on; // relay 4
%QX0.4 := cut_data.spindle;
//empty %QX0.5
//empty %QX0.6
//empty %QX0.7
%QX1.0 := supply_data.arm_clamp.on; // relay 5
%QX1.1 := supply_data.spindle_extract.on; // relay 6
%QX1.2 := work_data.alarm; // relay 7
%QX1.3 := FALSE; // relay 8
%QX1.4 := supply_data.feeder_small;
%QX1.5 := supply_data.feeder_linear;
%QX1.6 := supply_data.feeder_big;
//empty %QX1.7
//////////
//HMI UP//
//////////
IF hmi_data.hmi_ready THEN
	hmi_data.view_input_run := work_data.input_run.rise_physical.CLK;
	hmi_data.view_input_stop := work_data.input_stop.fall_physical.CLK;
	hmi_data.view_input_air := supply_data.input_air;
	hmi_data.view_input_hydraulic := supply_data.input_hydraulic;
	hmi_data.view_input_arm_clamp_holder_p := supply_data.input_arm_clamp_holder_p;
	hmi_data.view_input_feeder_small := supply_data.input_feeder_small;
	hmi_data.view_input_feeder_big := supply_data.input_feeder_big;
	hmi_data.view_input_jog_counter_a := %IX0.0;
	hmi_data.view_input_jog_counter_b := %IX0.1;
	hmi_data.view_input_jog_index_a := %IX1.0;
	hmi_data.view_input_jog_index_b := %IX1.1;
	hmi_data.view_input_spindle_encoder := %IX0.4;
	hmi_data.view_input_jog_index := work_data.input_jog_index;
	hmi_data.view_input_jog_micro := LREAL_TO_DINT(work_data.jog_encoder^.fActPosition * 1000);
	//
	hmi_data.view_output_arm_clamp_holder := supply_data.arm_clamp_holder.on;
	hmi_data.view_output_arm_clamp := supply_data.arm_clamp.on;
	hmi_data.view_output_spindle_clamp_n := supply_data.spindle_clamp_release;
	hmi_data.view_output_spindle_clamp_p := supply_data.spindle_clamp.on;
	hmi_data.view_output_spindle_extract := supply_data.spindle_extract.on;
	hmi_data.view_output_hydraulic := supply_data.hydraulic;
	hmi_data.view_output_alarm := work_data.alarm;
	hmi_data.view_output_spindle := cut_data.spindle;
	hmi_data.view_output_feeder_small := supply_data.feeder_small;
	hmi_data.view_output_feeder_linear := supply_data.feeder_linear;
	hmi_data.view_output_feeder_big := supply_data.feeder_big;
	//
	hmi_data.view_can_run := work_data.can_run;
	hmi_data.view_can_stop := work_data.can_stop;
	hmi_data.view_can_home := work_data.can_home;
	hmi_data.view_run_auto := work_data.run_auto.on;
	hmi_data.view_manual_active := work_data.manual_active;
	//
	hmi_data.view_overload := work_data.overload;
	hmi_data.view_cycle_count := cycle_count;
	hmi_data.view_cycle_time_msec := work_data.cycle_time_msec;
	//
	hmi_data.view_axiss_position_micron[0] := LREAL_TO_UDINT(cut_data.axiss[0].ref^.fActPosition);
	hmi_data.view_axiss_position_micron[1] := LREAL_TO_UDINT(cut_data.axiss[1].ref^.fActPosition);
	hmi_data.view_axiss_position_micron[2] := LREAL_TO_UDINT(supply_data.axis.ref^.fActPosition);
	hmi_data.view_axiss_torque_mNm[0] := LREAL_TO_UDINT(cut_data.axiss[0].torque_Nm_abs * 1E3);
	hmi_data.view_axiss_torque_mNm[1] := LREAL_TO_UDINT(cut_data.axiss[1].torque_Nm_abs * 1E3);
	hmi_data.view_axiss_torque_mNm[2] := LREAL_TO_UDINT(supply_data.axis.torque_Nm_abs * 1E3);
	//
	supply_data.foil_short_rise(CLK:= supply_data.foil_short, Q=> );
	IF supply_data.foil_short_rise.Q THEN
		hmi_data.view_supply_foil_short := TRUE;
	END_IF
	hmi_data.view_supply_foil_stuck := supply_data.foil_stuck;
	//
	hmi_data.view_cut_spindle_run_ing := cut_data.state_spindle = State.RUN_ING;
	hmi_data.view_cut_spindle_rpm := LREAL_TO_UDINT(ABS(cut_data.spindle_rps * 60));
	hmi_data.view_supply_test[0] := (work_data.can_run OR work_data.manual_active) AND supply_data.state_ready;
	hmi_data.view_supply_test[1] := (work_data.can_run OR work_data.manual_active) AND supply_data.state = 110;
	hmi_data.view_supply_test[2] := (work_data.can_run OR work_data.manual_active) AND supply_data.state = 120;
	hmi_data.view_supply_test[3] := (work_data.can_run OR work_data.manual_active) AND supply_data.state = 130;
	//
	hmi_data.view_state_work := work_data.state;
	hmi_data.view_state_supply := supply_data.state;
	hmi_data.view_state_cut := cut_data.state;
	hmi_data.view_state_cut_spindle := cut_data.state_spindle;
END_IF
END_ACTION

ACTION motion:
FOR i := 0 TO c_axis_i_max BY 1 DO
	axiss_read[i](
		xExecute:= , 
		xAbort:= , 
		uiIndex:= , 
		usiSubIndex:= , 
		Axis:= axiss[i]^, 
		xDone=> , 
		xBusy=> , 
		xError=> , 
		usiDataLength=> , 
		dwValue=> , 
		dwErrorCode=> , 
		eError=> );
	axiss_write[i](
		xExecute:= , 
		xAbort:= , 
		uiIndex:= , 
		usiSubIndex:= , 
		usiDataLength:= , 
		dwValue:= , 
		Axis:= axiss[i]^, 
		xDone=> , 
		xBusy=> , 
		xError=> , 
		dwErrorCode=> , 
		eError=> );
	axiss_read_status[i](
		Axis:= axiss[i]^, 
		Enable:= , 
		Valid=> , 
		Busy=> , 
		Error=> , 
		ErrorID=> , 
		Disabled=> , 
		Errorstop=> , 
		Stopping=> , 
		StandStill=> , 
		DiscreteMotion=> , 
		ContinuousMotion=> , 
		SynchronizedMotion=> , 
		Homing=> , 
		ConstantVelocity=> , 
		Accelerating=> , 
		Decelerating=> , 
		FBErrorOccured=> );
	axiss_set_mode[i](
		Axis:= axiss[i]^, 
		bExecute:= , 
		nControllerMode:= , 
		bDone=> , 
		bBusy=> , 
		bError=> , 
		nErrorID=> );
	axiss_power[i](
		Axis:= axiss[i]^,
		Enable:= , 
		bRegulatorOn:= , 
		bDriveStart:= , 
		Status=> , 
		bRegulatorRealState=> , 
		bDriveStartRealState=> , 
		Busy=> , 
		Error=> , 
		ErrorID=> );
	axiss_reset[i](
		Axis:= axiss[i]^,
		Execute:= ,
		Done=> ,
		Busy=> ,
		Error=> ,
		ErrorID=> );
	axiss_stop[i](
		Axis:= axiss[i]^, 
		Execute:= , 
		Deceleration:= , 
		Jerk:= , 
		Done=> , 
		Busy=> , 
		Error=> , 
		ErrorID=> );
	axiss_inch[i](
		Axis:= axiss[i]^, 
		InchForward:= , 
		InchBackward:= , 
		Distance:= , 
		Velocity:= , 
		Acceleration:= , 
		Deceleration:= , 
		Jerk:= , 
		Busy=> , 
		CommandAborted=> , 
		Error=> , 
		ErrorId=> );
	axiss_fsv[i](
		Axis:= axiss[i]^, 
		bExecute:= , 
		bAbort:= , 
		dwValueMask:= , 
		fSetPosition:= , 
		fSetVelocity:= , 
		fSetAcceleration:= , 
		fSetJerk:= , 
		fSetTorque:= , 
		fSetCurrent:= , 
		bBusy=> , 
		bCommandAborted=> , 
		bError=> , 
		iErrorID=> );
	axiss_sp[i](
		Axis:= axiss[i]^, 
		Execute:= , 
		Position:= , 
		Mode:= , 
		Done=> , 
		Busy=> , 
		Error=> , 
		ErrorID=> );
	axiss_mabs[i](
		Axis:= axiss[i]^, 
		Execute:= , 
		Position:= , 
		Velocity:= , 
		Acceleration:= , 
		Deceleration:= , 
		Jerk:= , 
		Direction:= , 
		BufferMode:= , 
		Done=> , 
		Busy=> , 
		Active=> , 
		CommandAborted=> , 
		Error=> , 
		ErrorID=> );
END_FOR
END_ACTION

ACTION save_check:
hmi_data.save_need := (
	save_data.supply_begin_micro_deg <> hmi_data.save_data.supply_begin_micro_deg OR
	save_data.supply_mid_micro_deg <> hmi_data.save_data.supply_mid_micro_deg OR
	save_data.supply_end_micro_deg <> hmi_data.save_data.supply_end_micro_deg OR
	save_data.supply_micro_deg_per_sec <> hmi_data.save_data.supply_micro_deg_per_sec OR
	//
	save_data.supply_arm_clamp_holder_n_delay_msec <> hmi_data.save_data.supply_arm_clamp_holder_n_delay_msec OR
	save_data.supply_arm_clamp_holder_p_delay_msec <> hmi_data.save_data.supply_arm_clamp_holder_p_delay_msec OR
	save_data.supply_arm_clamp_n_delay_msec <> hmi_data.save_data.supply_arm_clamp_n_delay_msec OR
	save_data.supply_arm_clamp_p_delay_msec <> hmi_data.save_data.supply_arm_clamp_p_delay_msec OR
	save_data.supply_spindle_clamp_n_delay_msec <> hmi_data.save_data.supply_spindle_clamp_n_delay_msec OR
	save_data.supply_spindle_clamp_p_delay_msec <> hmi_data.save_data.supply_spindle_clamp_p_delay_msec OR
	save_data.supply_spindle_extract_n_delay_msec <> hmi_data.save_data.supply_spindle_extract_n_delay_msec OR
	save_data.supply_spindle_extract_p_delay_msec <> hmi_data.save_data.supply_spindle_extract_p_delay_msec OR
	//
	save_data.cut_begin_micron[0] <> hmi_data.save_data.cut_begin_micron[0] OR
	save_data.cut_begin_micron[1] <> hmi_data.save_data.cut_begin_micron[1] OR
	save_data.cut_rapid_micron[0] <> hmi_data.save_data.cut_rapid_micron[0] OR
	save_data.cut_rapid_micron[1] <> hmi_data.save_data.cut_rapid_micron[1] OR
	save_data.cut_end_micron[0] <> hmi_data.save_data.cut_end_micron[0] OR
	save_data.cut_end_micron[1] <> hmi_data.save_data.cut_end_micron[1] OR
	save_data.cut_offset_micron[0] <> hmi_data.save_data.cut_offset_micron[0] OR
	save_data.cut_offset_micron[1] <> hmi_data.save_data.cut_offset_micron[1] OR
	//
	save_data.cut_lag_micron <> hmi_data.save_data.cut_lag_micron OR
	save_data.cut_rapid_micron_per_rev <> hmi_data.save_data.cut_rapid_micron_per_rev OR
	save_data.cut_micron_per_rev <> hmi_data.save_data.cut_micron_per_rev OR
	save_data.cut_dwell_msec <> hmi_data.save_data.cut_dwell_msec OR
	save_data.cut_retract_micron <> hmi_data.save_data.cut_retract_micron OR
	save_data.cut_retract_micron_per_sec <> hmi_data.save_data.cut_retract_micron_per_sec OR
	save_data.cut_spindle_encoder_resolution <> hmi_data.save_data.cut_spindle_encoder_resolution OR
	//
	save_data.home_encoder_value_recorded <> hmi_data.save_data.home_encoder_value_recorded OR
	save_data.home_encoder_value[0] <> hmi_data.save_data.home_encoder_value[0] OR
	save_data.home_encoder_value[1] <> hmi_data.save_data.home_encoder_value[1] OR
	save_data.home_encoder_value[2] <> hmi_data.save_data.home_encoder_value[2]
);
END_ACTION

ACTION save_apply:
/////////
//LIMIT//
/////////
save_data.supply_begin_micro_deg := MIN(c_supply_μdeg_max - 80_000, save_data.supply_begin_micro_deg);
save_data.supply_mid_micro_deg := MIN(c_supply_μdeg_max - 5_000, save_data.supply_mid_micro_deg);
save_data.supply_end_micro_deg := MIN(c_supply_μdeg_max, save_data.supply_end_micro_deg);
save_data.supply_micro_deg_per_sec := MIN(LREAL_TO_UDINT(c_supply_μdeg_per_sec_max), save_data.supply_micro_deg_per_sec);
//
save_data.supply_arm_clamp_holder_n_delay_msec := MAX(0_001, MIN(5_000, save_data.supply_arm_clamp_holder_n_delay_msec));
save_data.supply_arm_clamp_holder_p_delay_msec := MAX(0_001, MIN(5_000, save_data.supply_arm_clamp_holder_p_delay_msec));
save_data.supply_arm_clamp_n_delay_msec := MAX(0_001, MIN(5_000, save_data.supply_arm_clamp_n_delay_msec));
save_data.supply_arm_clamp_p_delay_msec := MAX(0_001, MIN(5_000, save_data.supply_arm_clamp_p_delay_msec));
save_data.supply_spindle_clamp_n_delay_msec := MAX(0_001, MIN(5_000, save_data.supply_spindle_clamp_n_delay_msec));
save_data.supply_spindle_clamp_p_delay_msec := MAX(0_001, MIN(5_000, save_data.supply_spindle_clamp_p_delay_msec));
save_data.supply_spindle_extract_n_delay_msec := MAX(0_001, MIN(5_000, save_data.supply_spindle_extract_n_delay_msec));
save_data.supply_spindle_extract_p_delay_msec := MAX(0_001, MIN(5_000, save_data.supply_spindle_extract_p_delay_msec));
//
save_data.cut_end_micron[0] := MAX(10_000, MIN(c_cut_stroke_μm, save_data.cut_end_micron[0]));
save_data.cut_end_micron[1] := MAX(10_000, MIN(c_cut_stroke_μm, save_data.cut_end_micron[1]));
save_data.cut_rapid_micron[0] := MIN(save_data.cut_end_micron[0] - 0_500, save_data.cut_rapid_micron[0]);
save_data.cut_rapid_micron[1] := MIN(save_data.cut_end_micron[1] - 0_500, save_data.cut_rapid_micron[1]);
save_data.cut_begin_micron[0] := MIN(save_data.cut_rapid_micron[0] - 0_500, save_data.cut_begin_micron[0]);
save_data.cut_begin_micron[1] := MIN(save_data.cut_rapid_micron[1] - 0_500, save_data.cut_begin_micron[1]);
save_data.cut_offset_micron[0] := MAX(-9_000, MIN(9_000, save_data.cut_offset_micron[0]));
save_data.cut_offset_micron[1] := MAX(-9_000, MIN(9_000, save_data.cut_offset_micron[1]));
//
save_data.cut_lag_micron := MAX(0_100, MIN(3_000, save_data.cut_lag_micron));
save_data.cut_rapid_micron_per_rev := MAX(0_001, MIN(1_000, save_data.cut_rapid_micron_per_rev));
save_data.cut_micron_per_rev := MAX(0_001, MIN(0_500, save_data.cut_micron_per_rev));
save_data.cut_dwell_msec := MAX(0_001, MIN(1_000, save_data.cut_dwell_msec));
save_data.cut_retract_micron_per_sec := MAX(5_000, MIN(LREAL_TO_UDINT(c_cut_μm_per_sec_max), save_data.cut_retract_micron_per_sec));
//
save_data.home_encoder_value[0] := MAX(0, MIN(cut_data.axiss[0].encoder_resolution - 1, save_data.home_encoder_value[0]));
save_data.home_encoder_value[1] := MAX(0, MIN(cut_data.axiss[1].encoder_resolution - 1, save_data.home_encoder_value[1]));
save_data.home_encoder_value[2] := MAX(0, MIN(supply_data.axis.encoder_resolution - 1, save_data.home_encoder_value[2]));
/////////
//APPLY//
/////////
cut_data.axiss[0].home_encoder_value_recorded := save_data.home_encoder_value_recorded;
cut_data.axiss[1].home_encoder_value_recorded := save_data.home_encoder_value_recorded;
supply_data.axis.home_encoder_value_recorded := save_data.home_encoder_value_recorded;
cut_data.axiss[0].home_encoder_value := ADR(save_data.home_encoder_value[0]);
cut_data.axiss[1].home_encoder_value := ADR(save_data.home_encoder_value[1]);
supply_data.axis.home_encoder_value := ADR(save_data.home_encoder_value[2]);
//
supply_data.axis.home_hit_timer.PT := INT_TO_TIME(1_000);
supply_data.axis.home_offset_absolute_μ := 5_000;
supply_data.axis.home_back_μ_per_sec := 5_000; // 1_000 μ = 1 độ
supply_data.axis.home_forward_μ_per_sec := 15_000;
supply_data.axis.max_μ := UDINT_TO_LREAL(c_supply_μdeg_max);
supply_data.axis.max_μ_per_sec := c_supply_μdeg_per_sec_max;
supply_data.axis.overload_timer.PT := INT_TO_TIME(0_500);
supply_data.axis.ramp_time_sec := 0.1;
supply_data.axis.jerk_factor := 10;
supply_data.begin_μdeg := UDINT_TO_LREAL(save_data.supply_begin_micro_deg);
supply_data.mid_μdeg := UDINT_TO_LREAL(save_data.supply_mid_micro_deg);
supply_data.end_μdeg := UDINT_TO_LREAL(save_data.supply_end_micro_deg);
supply_data.μdeg_per_sec := UDINT_TO_LREAL(save_data.supply_micro_deg_per_sec);
//
FOR i := 0 TO 1 BY 1 DO
	cut_data.axiss[i].home_hit_timer.PT := INT_TO_TIME(1_000);
	cut_data.axiss[i].home_offset_absolute_μ := 5_000;
	cut_data.axiss[i].home_back_μ_per_sec := 10_000;
	cut_data.axiss[i].home_forward_μ_per_sec := 30_000;
	cut_data.axiss[i].max_μ := UDINT_TO_LREAL(c_cut_stroke_μm);
	cut_data.axiss[i].max_μ_per_sec := c_cut_μm_per_sec_max;
	cut_data.axiss[i].overload_timer.PT := INT_TO_TIME(0_500);
	cut_data.axiss[i].ramp_time_sec := 0.1;
	cut_data.axiss[i].jerk_factor := 20;
	cut_data.begin_μm[i] := UDINT_TO_LREAL(save_data.cut_begin_micron[i]) + save_data.cut_offset_micron[i];
	cut_data.rapid_μm[i] := UDINT_TO_LREAL(save_data.cut_rapid_micron[i]) + save_data.cut_offset_micron[i];
	cut_data.end_μm[i] := UDINT_TO_LREAL(save_data.cut_end_micron[i]) + save_data.cut_offset_micron[i];
END_FOR
cut_data.lag_μm := UDINT_TO_LREAL(save_data.cut_lag_micron);
cut_data.rapid_μm_per_rev := UDINT_TO_LREAL(save_data.cut_rapid_micron_per_rev);
cut_data.μm_per_rev := UDINT_TO_LREAL(save_data.cut_micron_per_rev);
cut_data.dwell_timer.PT := UINT_TO_TIME(save_data.cut_dwell_msec);
cut_data.retract_μm := UDINT_TO_LREAL(save_data.cut_retract_micron);
cut_data.retract_μm_per_sec := UDINT_TO_LREAL(save_data.cut_retract_micron_per_sec);
cut_data.spindle_encoder_resolution := MAX(1, save_data.cut_spindle_encoder_resolution);
//
supply_data.arm_clamp_holder.n_timer.PT := UINT_TO_TIME(save_data.supply_arm_clamp_holder_n_delay_msec);
supply_data.arm_clamp_holder.p_timer.PT := UINT_TO_TIME(save_data.supply_arm_clamp_holder_p_delay_msec);
supply_data.arm_clamp.n_timer.PT := UINT_TO_TIME(save_data.supply_arm_clamp_n_delay_msec);
supply_data.arm_clamp.p_timer.PT := UINT_TO_TIME(save_data.supply_arm_clamp_p_delay_msec);
supply_data.spindle_clamp.n_timer.PT := UINT_TO_TIME(save_data.supply_spindle_clamp_n_delay_msec);
supply_data.spindle_clamp.p_timer.PT := UINT_TO_TIME(save_data.supply_spindle_clamp_p_delay_msec);
supply_data.spindle_extract.n_timer.PT := UINT_TO_TIME(save_data.supply_spindle_extract_n_delay_msec);
supply_data.spindle_extract.p_timer.PT := UINT_TO_TIME(save_data.supply_spindle_extract_p_delay_msec);
supply_data.feeder_small_on_timer.PT := INT_TO_TIME(1_000);
supply_data.feeder_small_off_timer.PT := INT_TO_TIME(3_000);
supply_data.foil_stuck_timer.PT := INT_TO_TIME(1_000);
supply_data.foil_stuck_fix_timer.PT := INT_TO_TIME(1_000);
//
work_data.input_run.timer.PT := INT_TO_TIME(0_300);
work_data.run_auto.timer.PT := INT_TO_TIME(3_000);
work_data.cut_spindle_run_timer.PT := INT_TO_TIME(1_000);
work_data.supply_test_timer.PT := INT_TO_TIME(0_300);
work_data.supply_hydraulic_timer.PT := INT_TO_TIME(0_300);
/////////
//FINAL//
/////////
hmi_data.save_data := save_data;
END_ACTION

ACTION work:
CASE work_data.state OF
	State.RST:
		supply_data.axis.overload_check := FALSE;
		cut_data.axiss[0].overload_check := FALSE;
		cut_data.axiss[1].overload_check := FALSE;
		supply_data.state := State.RST;
		cut_data.state := State.RST;
		cut_data.state_spindle := State.RST;
		work_data.jog_encoder_counter_set.xExecute := TRUE;
		work_data.manual_active := FALSE;
		work_data.alarm := FALSE;
		work_data.final_cycle_flag := FALSE;
		work_data.final_cycle := FALSE;
		StateNext(work_data.state);
	2:
		IF (
			supply_data.state = State.RST_DONE AND
			cut_data.state = State.RST_DONE AND
			cut_data.state_spindle = State.READY AND
			work_data.jog_encoder_counter_set.xDone
		) THEN
			work_data.state := State.RST_DONE;
		END_IF
	State.RST_DONE:
		//do nothing
	//////\\
	////\\\\
	//\\\\\\
	State.HOME:
		cut_data.state := State.HOME;
		StateNext(work_data.state);
	52:
		IF cut_data.state = State.HOME_DONE THEN
			supply_data.state := State.HOME;
			StateNext(work_data.state);
		END_IF
	53:
		IF supply_data.state = State.HOME_DONE THEN
			supply_data.axis.overload_check := TRUE;
			cut_data.axiss[0].overload_check := TRUE;
			cut_data.axiss[1].overload_check := TRUE;
			work_data.state := State.HOME_DONE;
		END_IF
	//
	State.HOME_DONE:
		supply_data.state := State.HOME_OFFSET;
		cut_data.state := State.HOME_OFFSET;
		StateNext(work_data.state);
	91:
		IF (
			supply_data.state = State.HOME_OFFSET_DONE AND
			cut_data.state = State.HOME_OFFSET_DONE
		) THEN
			work_data.state := State.HOME_OFFSET_DONE;
		END_IF
	State.HOME_OFFSET_DONE:
		supply_data.state := State.READY;
		cut_data.state := State.READY;
		work_data.state := State.READY;
		work_data.manual_active := TRUE;
		IF NOT save_data.home_encoder_value_recorded THEN
			save_data.home_encoder_value_recorded := TRUE;
			save_apply();
		END_IF
	//////\\
	////\\\\
	//\\\\\\
	State.READY:
		IF work_data.manual_active THEN
			CASE work_data.input_jog_index OF
				0: work_data.jog_i := ADR(cut_data.axiss[0]);
				1: work_data.jog_i := ADR(cut_data.axiss[1]);
				2: work_data.jog_i := ADR(supply_data.axis);
			END_CASE
			work_data.jog_i^.jog_delta := hmi_data.jog_micro_per_rev * (work_data.jog_encoder^.fActPosition - work_data.jog_encoder_last);
			work_data.jog_i^.jog_velocity := hmi_data.jog_micro_per_rev * work_data.jog_encoder^.fActVelocity;
			work_data.jog_i^.jog_acceleration := hmi_data.jog_micro_per_rev * work_data.jog_encoder^.fActAcceleration;
			work_data.jog_encoder_last := work_data.jog_encoder^.fActPosition;
		END_IF
	//////\\
	////\\\\
	//\\\\\\
	State.RUN:
		IF supply_data.state_ready AND cut_data.state_spindle = State.RUN_ING THEN
			supply_data.feeder_test := FALSE;
			work_data.manual_active := FALSE;
			supply_data.state := State.RUN;
			work_data.cycle_start_msec := time_msec;
			StateNext(work_data.state);
		END_IF
	102:
		IF supply_data.state = 110 THEN
			supply_data.state := 111;
			StateNext(work_data.state);
		END_IF
	103:
		IF supply_data.foil_stuck THEN
			work_data.alarm := TRUE;
		END_IF
		IF supply_data.state = 120 THEN
			cut_data.state := State.RUN;
			IF work_data.final_cycle THEN
				work_data.final_cycle := FALSE;
				supply_data.state := 141;
				work_data.state := 121;
			ELSE
				supply_data.state := 121;
				work_data.state := 111;
			END_IF
		END_IF
	//normal cycle
	111:
		IF supply_data.state = 130 THEN
			supply_data.state := 131;
			StateNext(work_data.state);
		END_IF
	112:
		IF cut_data.state = State.READY AND supply_data.state = 140 THEN
			work_data.state := 131;
		END_IF
	//final cycle
	121:
		IF cut_data.state = State.READY AND supply_data.state = 140 THEN
			supply_data.state := State.RUN; // extract foil
			StateNext(work_data.state);
		END_IF
	122:
		IF supply_data.state = 110 THEN
			supply_data.state := State.READY; // ready for rerun
			work_data.state := 131;
		END_IF
	//end
	131:
		work_data.state := State.READY;
		work_data.cycle_time_msec := ULINT_TO_UDINT(time_msec - work_data.cycle_start_msec);
		work_data.alarm := FALSE;
		IF (time_msec - cycle_count_reset_time_msec) > 86400_000 THEN
			cycle_count := 0;
			cycle_count_reset_time_msec := (time_msec / 86400_000) * 86400_000;
		END_IF
		cycle_count := cycle_count + 1;
END_CASE
END_ACTION

END_PROGRAM

// Device/Application/StateNext
FUNCTION StateNext
VAR_INPUT
	state: REFERENCE TO INT;
END_VAR
VAR
END_VAR

state := state + 1;

END_FUNCTION

// Device/Application/SupplyFB
FUNCTION_BLOCK SupplyFB
VAR_INPUT
	data: POINTER TO SupplyData;
END_VAR

////////
//MAIN//
////////
data^.state_ready := data^.state = State.READY OR data^.state = 140;
data^.axis_fb(data:= ); // data của hàm này đã được set ở hàm MAIN
data^.foil_stuck_timer(IN:= , PT:= , Q=> , ET=> );
data^.arm_clamp_holder_p_rise(CLK:= data^.input_arm_clamp_holder_p, Q=> );
CASE data^.state OF
	//////\\
	////\\\\
	//\\\\\\
	State.RST:
		data^.arm_clamp_holder.on := FALSE;
		data^.spindle_extract.on := FALSE;
		data^.feeder_small := FALSE;
		data^.feeder_linear := FALSE;
		data^.feeder_big := FALSE;
		data^.foil_stuck := FALSE;
		StateNext(data^.state);
	2:
		IF (
			data^.arm_clamp_holder.n_timer.Q AND
			data^.spindle_extract.n_timer.Q
		) THEN
			data^.axis.state := State.RST;
			StateNext(data^.state);
		END_IF
	3:
		IF data^.axis.state = State.RST_DONE THEN
			data^.state := State.RST_DONE;
		END_IF
	//////\\
	////\\\\
	//\\\\\\
	State.HOME:
		data^.arm_clamp.on := FALSE;
		data^.spindle_clamp.on := FALSE;
		StateNext(data^.state);
	52:
		IF (
			data^.arm_clamp.n_timer.Q AND
			data^.spindle_clamp.n_timer.Q
		) THEN
			data^.axis.state := State.HOME;
			StateNext(data^.state);
		END_IF
	53:
		IF data^.axis.state = State.HOME_DONE THEN
			data^.state := State.HOME_DONE;
		END_IF
	//////\\
	////\\\\
	//\\\\\\
	State.HOME_OFFSET:
		data^.axis.home_offset_μ := data^.begin_μdeg;
		data^.axis.state := State.HOME_OFFSET;
		StateNext(data^.state);
	92:
		IF data^.axis.state = State.HOME_OFFSET_DONE THEN
			data^.axis.state := State.READY;
			data^.feeder_small := TRUE;
			data^.feeder_linear := TRUE;
			data^.feeder_big := TRUE;
			data^.state := State.HOME_OFFSET_DONE;
		END_IF
	State.READY:
		//do nothing
	//////\\
	////\\\\
	//\\\\\\
	// thoát phôi
	State.RUN:
		data^.arm_clamp_holder.on := FALSE; // make sure collision free move
		StateNext(data^.state);
	102:
		IF data^.arm_clamp_holder.n_timer.Q THEN
			data^.spindle_clamp.on := FALSE;
			StateNext(data^.state);
		END_IF
	103:
		IF data^.spindle_clamp.n_timer.Q THEN
			data^.spindle_extract.on := TRUE;
			StateNext(data^.state);
		END_IF
	104:
		IF data^.spindle_extract.p_timer.Q THEN
			data^.spindle_extract.on := FALSE;
			StateNext(data^.state);
		END_IF
	105:
		IF data^.spindle_extract.n_timer.Q THEN
			data^.state := 110;
		END_IF
	// cấp phôi
	111:
		data^.arm_clamp_holder.on := FALSE; // make sure collision free move
		data^.foil_stuck_timer.IN := FALSE;
		StateNext(data^.state);
	112:
		IF data^.arm_clamp_holder.n_timer.Q AND data^.axis.state = State.READY THEN
			data^.axis.target_position_μ := data^.end_μdeg;
			data^.axis.target_velocity_μ_per_sec := data^.μdeg_per_sec;
			data^.axis.state := State.RUN;
			StateNext(data^.state);
		END_IF
	113:
		IF data^.axis.state = State.READY THEN
			data^.arm_clamp_holder.on := TRUE;
			data^.foil_stuck_timer.IN := TRUE;
			StateNext(data^.state);
		END_IF
	114:
		IF data^.foil_stuck_timer.Q THEN
			data^.foil_stuck := TRUE;
			data^.foil_stuck_timer.IN := FALSE;
			data^.state := 141;
		END_IF
		IF data^.arm_clamp_holder_p_rise.Q THEN
			data^.spindle_clamp.on := TRUE;
			StateNext(data^.state);
		END_IF
	115:
		IF data^.spindle_clamp.p_timer.Q THEN
			data^.arm_clamp.on := FALSE;
			StateNext(data^.state);
		END_IF
	116:
		IF data^.arm_clamp.n_timer.Q THEN
			data^.arm_clamp_holder.on := FALSE;
			StateNext(data^.state);
		END_IF
	117:
		IF data^.arm_clamp_holder.n_timer.Q THEN
			data^.foil_stuck := FALSE;
			data^.state := 120;
		END_IF
	// lấy phôi mới
	121:
		data^.arm_clamp_holder.on := FALSE; // make sure collision free move
		StateNext(data^.state);
	122:
		IF data^.arm_clamp_holder.n_timer.Q AND data^.axis.state = State.READY THEN
			data^.axis.target_position_μ := data^.begin_μdeg;
			data^.axis.target_velocity_μ_per_sec := data^.μdeg_per_sec;
			data^.axis.state := State.RUN;
			StateNext(data^.state);
		END_IF
	123:
		IF data^.axis.state = State.READY THEN
			data^.feeder_linear := FALSE;
			data^.arm_clamp_holder.on := TRUE;
			StateNext(data^.state);
		END_IF
	124:
		IF data^.arm_clamp_holder.p_timer.Q THEN
			data^.arm_clamp.on := TRUE;
			StateNext(data^.state);
		END_IF
	125:
		IF data^.arm_clamp.p_timer.Q THEN
			data^.arm_clamp_holder.on := FALSE;
			StateNext(data^.state);
		END_IF
	126:
		IF data^.arm_clamp_holder.n_timer.Q THEN
			data^.feeder_linear := TRUE;
			data^.state := 130;
		END_IF
	// di chuyển đến vị trí chờ
	131:
		data^.arm_clamp_holder.on := FALSE; // make sure collision free move
		StateNext(data^.state);
	132:
		IF data^.arm_clamp_holder.n_timer.Q AND data^.axis.state = State.READY THEN
			data^.axis.target_position_μ := data^.mid_μdeg;
			data^.axis.target_velocity_μ_per_sec := data^.μdeg_per_sec;
			data^.axis.state := State.RUN;
			StateNext(data^.state);
		END_IF
	133:
		IF data^.axis.state = State.READY THEN
			data^.state := 140;
		END_IF
	// di chuyển đến vị trí nghỉ
	141:
		data^.arm_clamp_holder.on := FALSE; // make sure collision free move
		StateNext(data^.state);
	142:
		IF data^.arm_clamp_holder.n_timer.Q AND data^.axis.state = State.READY THEN
			data^.axis.target_position_μ := data^.begin_μdeg;
			data^.axis.target_velocity_μ_per_sec := data^.μdeg_per_sec;
			data^.axis.state := State.RUN;
			StateNext(data^.state);
		END_IF
	143:
		IF data^.axis.state = State.READY THEN
			data^.state := 140;
		END_IF
END_CASE
//////////
//FEEDER//
//////////
data^.feeder_small_on_timer(IN:= NOT data^.input_feeder_small, PT:= , Q=> , ET=> );
data^.feeder_small_off_timer(IN:= data^.input_feeder_small, PT:= , Q=> , ET=> );
IF data^.state >= State.READY AND NOT data^.feeder_test THEN
	IF data^.feeder_small_on_timer.Q THEN
		data^.feeder_small := TRUE;
	END_IF
	IF data^.feeder_small_off_timer.Q THEN
		data^.feeder_small := FALSE;
	END_IF
END_IF

END_FUNCTION_BLOCK

// Device/Application/CutFB
FUNCTION_BLOCK CutFB
VAR_INPUT
	data: POINTER TO CutData;
END_VAR

VAR CONSTANT
	c_stable_cycle_valid: INT := 2;
END_VAR

////////
//MAIN//
////////
data^.axiss_fb[0](data:= ); // data của hàm này đã được set ở hàm MAIN
data^.axiss_fb[1](data:= );
data^.dwell_timer(IN:= , PT:= , Q=> , ET=> );
IF data^.time_msec - data^.spindle_encoder_time_msec_last >= 2_000 THEN
	data^.time_delta_sec := ULINT_TO_LREAL(data^.time_msec - data^.spindle_encoder_time_msec_last) * 1E-3;
	data^.spindle_rps := (
			DINT_TO_LREAL(data^.spindle_encoder_counter.diValue - data^.spindle_encoder_counter_last) / data^.spindle_encoder_resolution
		) / data^.time_delta_sec;
	data^.spindle_rps := MIN(3000 / 60, data^.spindle_rps);
	data^.spindle_encoder_counter_last := data^.spindle_encoder_counter.diValue;
	data^.spindle_encoder_time_msec_last := data^.time_msec;
	IF data^.spindle_rps - data^.spindle_rps_last < 0.5 THEN
		data^.spindle_rps_stable_cycle := MIN(data^.spindle_rps_stable_cycle + 1, c_stable_cycle_valid);
	ELSE
		data^.spindle_rps_stable_cycle := MAX(0, data^.spindle_rps_stable_cycle - 1);
	END_IF
	data^.spindle_rps_last := data^.spindle_rps;
END_IF
CASE data^.state OF
	//////\\
	////\\\\
	//\\\\\\
	State.RST:
		data^.axiss[0].state := State.RST;
		data^.axiss[1].state := State.RST;
		StateNext(data^.state);
	2:
		IF (
			data^.axiss[0].state = State.RST_DONE AND
			data^.axiss[1].state = State.RST_DONE
		)
		THEN
			data^.state := State.RST_DONE;
		END_IF
	//////\\
	////\\\\
	//\\\\\\
	State.HOME:
		data^.axiss[0].state := State.HOME;
		data^.axiss[1].state := State.HOME;
		StateNext(data^.state);
	52:
		IF (
			data^.axiss[0].state = State.HOME_DONE AND
			data^.axiss[1].state = State.HOME_DONE
		) THEN
			data^.state := State.HOME_DONE;
		END_IF
	//////\\
	////\\\\
	//\\\\\\
	State.HOME_OFFSET:
		data^.axiss[0].home_offset_μ := data^.retract_μm;
		data^.axiss[1].home_offset_μ := data^.retract_μm;
		data^.axiss[0].state := State.HOME_OFFSET;
		data^.axiss[1].state := State.HOME_OFFSET;
		StateNext(data^.state);
	92:
		IF (
			data^.axiss[0].state = State.HOME_OFFSET_DONE AND
			data^.axiss[1].state = State.HOME_OFFSET_DONE
		) THEN
			data^.axiss[0].state := State.READY;
			data^.axiss[1].state := State.READY;
			data^.state := State.HOME_OFFSET_DONE;
		END_IF
	//////\\
	////\\\\
	//\\\\\\
	State.READY:
		//do nothing
	//////\\
	////\\\\
	//\\\\\\
	State.RUN:
		IF (
			data^.axiss[0].state = State.READY AND
			data^.axiss[1].state = State.READY
		) THEN
			data^.axiss[0].target_position_μ := data^.retract_μm;
			data^.axiss[0].target_velocity_μ_per_sec := data^.retract_μm_per_sec;
			data^.axiss[0].state := State.RUN;
			data^.axiss[1].target_position_μ := data^.retract_μm;
			data^.axiss[1].target_velocity_μ_per_sec := data^.retract_μm_per_sec;
			data^.axiss[1].state := State.RUN;
			data^.dwell_timer.IN := FALSE;
			StateNext(data^.state);
		END_IF
	102:
		IF (
			data^.axiss[0].state = State.READY AND
			data^.axiss[1].state = State.READY
		) THEN
			data^.axiss[0].target_position_μ := data^.begin_μm[0];
			data^.axiss[0].target_velocity_μ_per_sec := data^.retract_μm_per_sec;
			data^.axiss[0].state := State.RUN;
			data^.axiss[1].target_position_μ := data^.begin_μm[1];
			data^.axiss[1].target_velocity_μ_per_sec := data^.retract_μm_per_sec;
			data^.axiss[1].state := State.RUN;
			StateNext(data^.state);
		END_IF
	103:
		IF (
			data^.axiss[0].state = State.READY AND
			data^.axiss[1].state = State.READY
		) THEN
			data^.axiss[0].target_position_μ := data^.rapid_μm[0]; // đã có giới hạn trong AxisLinearFB nên không cần giới hạn ở đây
			data^.axiss[0].target_velocity_μ_per_sec := data^.rapid_μm_per_rev * data^.spindle_rps;
			data^.axiss[0].state := State.RUN;
			StateNext(data^.state);
		END_IF
	104:
		IF (data^.axiss[0].ref^.fActPosition - data^.begin_μm[0]) >= data^.lag_μm OR data^.axiss[0].state = State.READY THEN
			data^.axiss[1].target_position_μ := data^.rapid_μm[1];
			data^.axiss[1].target_velocity_μ_per_sec := data^.rapid_μm_per_rev * data^.spindle_rps;
			data^.axiss[1].state := State.RUN;
			StateNext(data^.state);
		END_IF
	105:
		IF (
			data^.axiss[0].state = State.READY AND
			data^.axiss[1].state = State.READY
		) THEN
			data^.axiss[0].target_position_μ := data^.end_μm[0];
			data^.axiss[0].target_velocity_μ_per_sec := data^.μm_per_rev * data^.spindle_rps;
			data^.axiss[0].state := State.RUN;
			StateNext(data^.state);
		END_IF
	106:
		IF (data^.axiss[0].ref^.fActPosition - data^.rapid_μm[0]) >= data^.lag_μm OR data^.axiss[0].state = State.READY THEN
			data^.axiss[1].target_position_μ := data^.end_μm[1];
			data^.axiss[1].target_velocity_μ_per_sec := data^.μm_per_rev * data^.spindle_rps;
			data^.axiss[1].state := State.RUN;
			StateNext(data^.state);
		END_IF
	107:
		IF (
			data^.axiss[0].state = State.READY AND
			data^.axiss[1].state = State.READY
		) THEN
			data^.dwell_timer.IN := TRUE;
			StateNext(data^.state);
		END_IF
	108:
		IF data^.dwell_timer.Q THEN
			data^.axiss[0].target_position_μ := data^.retract_μm;
			data^.axiss[0].target_velocity_μ_per_sec := data^.retract_μm_per_sec;
			data^.axiss[0].state := State.RUN;
			data^.axiss[1].target_position_μ := data^.retract_μm;
			data^.axiss[1].target_velocity_μ_per_sec := data^.retract_μm_per_sec;
			data^.axiss[1].state := State.RUN;
			StateNext(data^.state);
		END_IF
	109:
		IF (
			data^.axiss[0].state = State.READY AND
			data^.axiss[1].state = State.READY
		) THEN
			data^.state := State.READY;
		END_IF
END_CASE
///////////
//SPINDLE//
///////////
CASE data^.state_spindle OF
	State.RST:
		data^.spindle := FALSE;
		data^.spindle_rps_stable_cycle := 0;
	 	StateNext(data^.state_spindle);
	2:
		data^.state_spindle := State.READY;
	//////\\
	////\\\\
	//\\\\\\
	State.READY:
		//do nothing
	//////\\
	////\\\\
	//\\\\\\
	State.RUN:
		data^.spindle := TRUE;
		data^.spindle_rps_stable_cycle := 0;
		StateNext(data^.state_spindle);
	102:
		IF data^.spindle_rps > 10 AND data^.spindle_rps_stable_cycle = c_stable_cycle_valid THEN
			data^.state_spindle := State.RUN_ING;
		END_IF
	//////\\
	////\\\\
	//\\\\\\
	State.RUN_ING:
		//check
END_CASE

END_FUNCTION_BLOCK

// Device/Application/AxisFB
FUNCTION_BLOCK PUBLIC AxisFB
VAR_INPUT
	data: POINTER TO AxisEC;
END_VAR

data^.torque_Nm := data^.ref^.fActTorque;
data^.torque_Nm_abs := ABS(data^.torque_Nm);
// giá trị .fActTorque có thể khác nhau tuỳ PLC, trong trường hợp PLC Inovance này fActTorque là giá trị từ phần trăm moment
// 0.0% đến hơn 100.0%, nên phải nhân với .torque_rated_Nm đọc được ở hàm MAIN
data^.home_hit_timer(IN:= , PT:= , Q=> , ET=> );
// timer để lấy gốc, khi lùi về chạm gốc, giá trị moment sẽ tăng lên đến giá trị quy định (trong chương trình này là 1.27Nm)
// để tránh bị nhiễu thì moment quy định cần phải duy trì trong một thời gian mới có thể xác định gốc
data^.overload_timer(IN:= , PT:= , Q=> , ET=> );
// timer quá tải
IF data^.overload_check THEN
	data^.overload_timer.IN := data^.torque_Nm_abs > (1.0 * data^.torque_rated_Nm);
	data^.overload := data^.overload_timer.Q OR data^.torque_Nm_abs > (3.0 * data^.torque_rated_Nm);
END_IF
//////\\
////\\\\
//\\\\\\
CASE data^.state OF
	State.RST: // reset trục
		data^.read_status^.Enable := TRUE; // bật đọc trạng thái servo
		StateNext(data^.state);
	2:
		IF data^.read_status^.Valid THEN
			StateNext(data^.state);
		END_IF
	3:
		data^.inch^.InchBackward := FALSE;
		data^.inch^.InchForward := FALSE;
		data^.fsv^.bExecute := FALSE;
		data^.fsv^.fSetPosition := data^.ref^.fActPosition;
		StateNext(data^.state);
	4:
		IF NOT data^.inch^.Busy AND NOT data^.fsv^.bError THEN
			StateNext(data^.state);
		END_IF
	5:
		IF data^.mabs^.Busy THEN // nếu hàm dịch chuyển MC_MoveAbsolute đang hoạt dộng thì kích hoạt hàm MC_Stop
			data^.stop^.Deceleration := data^.mabs^.Velocity / 0.1;
			data^.stop^.Jerk := data^.stop^.Deceleration * data^.jerk_factor;
			data^.stop^.Execute := TRUE;
			StateNext(data^.state);
		ELSE // nếu không thì nhảy đến bước tiếp theo
			data^.state := 21;
		END_IF
	6: // hàm SMC_Inch đang không hoạt động và hàm MC_Stop hoàn thành
		IF data^.stop^.Done THEN
			data^.state := 21;
		END_IF
	//
	21:
		data^.mabs^.Execute := FALSE; // sau khi các hàm hoàn thành, phải đặt biến Execute về FALSE
		data^.stop^.Execute := FALSE; // vì muốn chạy hàm cần có tín hiệu rising edge
		data^.power^.bDriveStart := FALSE; // tắt servo
		StateNext(data^.state);
	22:
		IF NOT data^.power^.Status THEN // đã tắt xong servo
			StateNext(data^.state);
		END_IF
	23:
		IF data^.read_status^.FBErrorOccured THEN // nếu có lỗi xảy ra thì xoá lỗi cũ
			SMC_ClearFBError(pDrive:= data^.ref); // xoá lỗi
			StateNext(data^.state);
		ELSE // nếu không có thì nhảy đến bước cuối
			data^.state := 31;
		END_IF
	24:
		IF data^.read_status^.FBErrorOccured THEN
			data^.reset^.Execute := TRUE; // reset lỗi
			StateNext(data^.state);
		END_IF
	25:
		IF data^.reset^.Done THEN
			data^.reset^.Execute := FALSE;
			SMC_ClearFBError(pDrive:= data^.ref); // xoá lỗi
			data^.state := 31;
		END_IF
	//
	31:
		data^.read_status^.Enable := FALSE;
		data^.state := State.RST_DONE;
	//////\\
	////\\\\
	//\\\\\\
	State.HOME:
		data^.power^.bDriveStart := TRUE; // bật servo để bắt đầu lấy gốc
		StateNext(data^.state);
	52:
		IF data^.power^.Status THEN // servo đã sẵn sàng
			StateNext(data^.state);
		END_IF
	53:
		IF data^.home_done THEN // đã lấy gốc trước đó thì nhảy đến bước HOME_FORWARD
			data^.state := State.HOME_FORWARD;
		ELSE // chưa lấy gốc thì qua bước tiếp theo
			StateNext(data^.state);
		END_IF
	54:
		data^.set_mode^.nControllerMode := SMC_CONTROLLER_MODE.SMC_velocity;// chuyển chế độ servo sang tốc độ
		// ở chế độ .SMC_torque hoặc .SMC_velocity, khi servo vị chặn nó sẽ không vọt sau khi được nhả ra
		data^.set_mode^.bExecute := TRUE;
		StateNext(data^.state);
	55:
		IF data^.set_mode^.bDone THEN // chuyển chế độ xong
			data^.set_mode^.bExecute := FALSE;
			StateNext(data^.state);
		END_IF
	56:
		data^.home_torque_Nm := MIN(1.27, data^.torque_rated_Nm);
		IF data^.ref^.fScalefactor > 0 THEN
			data^.write^.uiIndex := 16#60E1; // servo negative torque limit
		ELSE
			data^.write^.uiIndex := 16#60E0; // servo positive torque limit
		END_IF
		data^.write^.usiSubIndex := 0;
		data^.write^.usiDataLength := 2;
		data^.write^.dwValue := LREAL_TO_DWORD(1000 * (data^.home_torque_Nm / data^.torque_rated_Nm));
		data^.write^.xExecute := TRUE;
		// đặt giá trị moment, 1.27Nm là tối đa, với vít me bước 5mm thì lực ép ở 1.27Nm sẽ là (1.27*2*PI)/0.005 = 1595N
		// khoảng 160 kg
		// moment không được vượt quá moment danh định vì nó sẽ lỗi quá tải khi ngâm ở thời gian dài với home_hit_timer
		// thực thi hàm limit_torque
		// hãy đọc function defination của hàm này
		// tuỳ servo mà 100% = 1000
		StateNext(data^.state);
	57:
		IF data^.write^.xDone THEN // set xong giới hạn moment
			data^.write^.xExecute := FALSE;
			StateNext(data^.state);
		END_IF
	58:
		data^.inch^.Velocity := data^.home_back_μ_per_sec; // lùi về
		data^.inch^.Distance := 500_000; // hàm SMC_Inch có giới hạn bới .Distance, khác với hàm MC_Jog không có giới hạn
		// đặt .Distance = 500_000 hay số nào đó thật lớn cũng được
		data^.inch^.Acceleration := data^.inch^.Velocity / 0.1;
		data^.inch^.Deceleration := data^.inch^.Acceleration;
		data^.inch^.Jerk := data^.inch^.Acceleration * data^.jerk_factor;
		data^.inch^.InchBackward := TRUE; // .InchBackward là lùi
		data^.inch^.InchForward := FALSE; // .InchForward là tiến
		// nếu .InchBackward và .InchForward cùng bằng TRUE hoặc FALSE thì servo không chạy
		data^.home_hit_timer.IN := FALSE; // reset timer
		StateNext(data^.state);
	59:
		data^.home_hit_timer.IN := ABS(data^.torque_Nm) >= data^.home_torque_Nm * 0.95; // set timer, * 0.95 để chắc ăn, tránh bị nhiễu
		IF data^.home_hit_timer.Q THEN // khi timer kích hoạt, dừng hàm SMC_Inch
			data^.inch^.InchBackward := FALSE;
			data^.inch^.InchForward := FALSE;
			data^.mabs^.Position := data^.ref^.fActPosition + data^.home_offset_absolute_μ;
			IF data^.home_encoder_value_recorded THEN
				data^.home_encoder_delta := data^.home_encoder_value^ - data^.encoder_single_position;
				IF data^.home_encoder_delta >= 0 THEN
					data^.home_delta_μ := ABS(data^.home_encoder_delta) / data^.ref^.fScalefactor;
				ELSIF ABS(data^.home_encoder_delta) > (data^.encoder_resolution / 2) THEN
					data^.home_delta_μ := (data^.encoder_resolution - ABS(data^.home_encoder_delta)) / data^.ref^.fScalefactor;
				ELSE
					data^.home_delta_μ := -ABS(data^.home_encoder_delta) / data^.ref^.fScalefactor;
				END_IF
				data^.mabs^.Position := data^.mabs^.Position + data^.home_delta_μ;
			ELSE
				data^.home_encoder_value^ := data^.encoder_single_position;
				data^.home_encoder_value_recorded := TRUE;
			END_IF
			// gán tạm giá trị vào hàm MC_MoveAbsolute để đến bước tiếp theo
			// .fActPosition là vị trí thực tế của servo
			// ví dụ .fActPosition khi chạm là -123_000, có thể dùng "_" để phân cách các con số cho dễ đọc
			// .home_offset_absolute_micron = 1_000
			// data^.mabs^.Position sẽ bằng -123_000 + 1_000 = -122_000
			StateNext(data^.state);
		END_IF
	60:
		data^.sp^.Position := data^.ref^.fActPosition - data^.mabs^.Position;
		// thực hiện hàm MC_SetPosition để đưa giá trị .fActPosition về 0
		// bây giờ giá trị data^.sp^.Position = -123_000 - (-122_000) = -1_000
		// bây giờ servo đang ở vị trí va chạm, để về gốc thì nó phải dịch chuyển 1_000 micron
		// vậy vị trí gốc cách vị trí va chạm đúng bằng .home_offset_absolute_micron
		data^.sp^.Execute := TRUE;
		StateNext(data^.state);
	61:
		IF data^.sp^.Done THEN // set xong tiến tới HOME_FORWARD
			data^.sp^.Execute := FALSE;
			data^.state := State.HOME_FORWARD;
			data^.home_done := TRUE;
		END_IF
	//////\\
	////\\\\
	//\\\\\\
	State.HOME_FORWARD:
		IF NOT data^.inch^.Busy THEN
			data^.set_mode^.nControllerMode := SMC_CONTROLLER_MODE.SMC_position; // set mode về điều khiển vị trí
			data^.set_mode^.bExecute := TRUE;
			StateNext(data^.state);
		END_IF
	72:
		IF data^.set_mode^.bDone THEN
			data^.set_mode^.bExecute := FALSE;
			StateNext(data^.state);
		END_IF
	73:
		IF data^.ref^.fScalefactor > 0 THEN
			data^.write^.uiIndex := 16#60E1; // servo negative torque limit
		ELSE
			data^.write^.uiIndex := 16#60E0; // servo positive torque limit
		END_IF
		data^.write^.usiSubIndex := 0;
		data^.write^.usiDataLength := 2;
		data^.write^.dwValue := DINT_TO_DWORD(3000);
		data^.write^.xExecute := TRUE;
		StateNext(data^.state);
		// đưa giới hạn moment về 300%
	74:
		IF data^.write^.xDone THEN
			data^.write^.xExecute := FALSE;
			StateNext(data^.state);
		END_IF
	75:
		// dịch chuyển tới vị trí gốc
		data^.mabs^.Position := 0;
		data^.mabs^.Velocity := data^.home_forward_μ_per_sec;
		data^.mabs^.Acceleration := data^.mabs^.Velocity / data^.ramp_time_sec;
		data^.mabs^.Deceleration := data^.mabs^.Acceleration;
		data^.mabs^.Jerk := data^.mabs^.Acceleration * data^.jerk_factor;
		data^.mabs^.Execute := TRUE;
		StateNext(data^.state);
	76:
		IF data^.mabs^.Done THEN
			data^.mabs^.Execute := FALSE;
			data^.state := State.HOME_DONE;
		END_IF
	//////\\
	////\\\\
	//\\\\\\
	State.HOME_OFFSET: // địch chuyển tới vị trí HOME_OFFSET
		data^.mabs^.Position := data^.home_offset_μ;
		data^.mabs^.Velocity := data^.home_forward_μ_per_sec;
		data^.mabs^.Acceleration := data^.mabs^.Velocity / data^.ramp_time_sec;
		data^.mabs^.Deceleration := data^.mabs^.Acceleration;
		data^.mabs^.Jerk := data^.mabs^.Acceleration * data^.jerk_factor; // jerk chỉ có tác dụng khi Velocity ramp type khác Trapezoid
		data^.mabs^.Execute := TRUE;
		StateNext(data^.state);
	92:
		IF data^.mabs^.Done THEN // dịch chuyển xong
			data^.mabs^.Execute := FALSE;
			StateNext(data^.state);
		END_IF
	93:
		data^.jog_delta := 0;
		data^.fsv^.dwValueMask := UDINT_TO_DWORD(1 + 2 + 4 + 8);
		data^.fsv^.fSetPosition := data^.home_offset_μ;
		data^.fsv^.fSetVelocity := 0;
		data^.fsv^.fSetAcceleration := 0;
		data^.fsv^.fSetJerk := 0;
		data^.fsv^.bExecute := TRUE;
		data^.state := State.HOME_OFFSET_DONE;
	//////\\
	////\\\\
	//\\\\\\
	State.READY:
		IF data^.fsv^.bExecute AND NOT data^.fsv^.bError THEN
			data^.fsv^.fSetPosition := MAX(0, MIN(data^.max_μ, data^.fsv^.fSetPosition + data^.jog_delta));
			data^.fsv^.fSetVelocity := MIN(data^.max_μ_per_sec, ABS(data^.jog_velocity));
			data^.fsv^.fSetAcceleration := MIN(data^.max_μ_per_sec * 10, ABS(data^.jog_acceleration));
			data^.fsv^.fSetJerk := data^.fsv^.fSetAcceleration * data^.jerk_factor;
		END_IF
		data^.jog_delta := 0;
	//////\\
	////\\\\
	//\\\\\\
	State.RUN:
		IF data^.fsv^.bExecute THEN
			data^.fsv^.bExecute := FALSE;
			StateNext(data^.state);
		ELSE
			data^.state := 103;
		END_IF
	102:
		IF NOT data^.fsv^.bError THEN
			StateNext(data^.state);
		END_IF
	103:
		// lệnh chạy đến vị trí chỉ định
		// xem hàm cut() và supply()
		// set data^.target_position_micron và data^.target_velocity_micron_per_sec sau đó set data^.state = State.RUN
		data^.mabs^.Position := MAX(0, MIN(data^.max_μ, data^.target_position_μ)); // giới hạn vị trí, xem save_apply()
		data^.mabs^.Velocity := MAX(0_100, MIN(data^.max_μ_per_sec, data^.target_velocity_μ_per_sec)); // giới hạn tốc độ, xem save_apply()
		data^.mabs^.Acceleration := data^.mabs^.Velocity / data^.ramp_time_sec;
		data^.mabs^.Deceleration := data^.mabs^.Acceleration;
		data^.mabs^.Jerk := data^.mabs^.Acceleration * data^.jerk_factor;
		data^.mabs^.Execute := TRUE;
		StateNext(data^.state);
	104:
		IF data^.mabs^.Done THEN
			data^.mabs^.Execute := FALSE;
			data^.state := State.READY;
		END_IF
END_CASE

END_FUNCTION_BLOCK

// Device/Application/Visualization
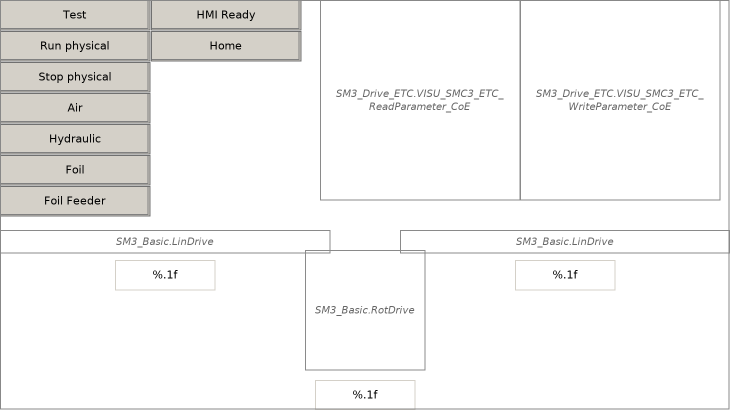
VISUALIZATION Visualization  // 730x410
    Button (0,31 150x30), "Run physical"
        toggle MAIN.work_data.input_run.rise_physical.CLK
    Frame (305,250 120x120)
        shows SM3_Basic.RotDrive(m_Input_AXISREF := MAIN.axiss[2]^)
    Frame (0,230 330x23)
        shows SM3_Basic.LinDrive(m_Input_AXISREF := MAIN.axiss[0]^)
    Frame (400,230 330x23)
        shows SM3_Basic.LinDrive(m_Input_AXISREF := MAIN.axiss[1]^)
    Button (0,0 150x30), "Test"
        toggle MAIN.test
    Button (0,62 150x30), "Stop physical"
        toggle MAIN.work_data.input_stop.fall_physical.CLK
    Button (0,93 150x30), "Air"
        toggle MAIN.supply_data.input_air
    Button (0,124 150x30), "Hydraulic"
        toggle MAIN.supply_data.input_hydraulic
    Button (151,0 150x30), "HMI Ready"
        toggle MAIN.hmi_data.hmi_ready
    Button (151,31 150x30), "Home"
        toggle MAIN.hmi_data.home
    Textfield (115,260 100x30), "%.1f", text variable: MAIN.cut_data.axiss[0].home_delta_μ
    Textfield (515,260 100x30), "%.1f", text variable: MAIN.cut_data.axiss[1].home_delta_μ
    Textfield (315,380 100x30), "%.1f", text variable: MAIN.supply_data.axis.home_delta_μ
    Button (0,155 150x30), "Foil"
        toggle MAIN.supply_data.input_foil
    Frame (320,0 200x200)
        shows SM3_Drive_ETC.VISU_SMC3_ETC_ReadParameter_CoE(m_Input_FB := MAIN.axiss_read[0])
    Frame (520,0 200x200)
        shows SM3_Drive_ETC.VISU_SMC3_ETC_WriteParameter_CoE(m_Input_FB := MAIN.axiss_write[0])
    Button (0,186 150x30), "Foil Feeder"
        toggle MAIN.supply_data.input_foil_feeder
END_VISUALIZATION
